// SIMATIC S7-200 SMART project (STEP 7-Micro/WIN SMART), CPU ST20

SYMBOL_TABLE 系统符号
Always_On        SM0.0    // 始终接通
First_Scan_On    SM0.1    // 仅在第一个扫描周期时接通
END_SYMBOL_TABLE

ORGANIZATION_BLOCK MAIN:OB1
TITLE=// ============================================================
// // 文件: OB1_MAIN.stl
// // 功能: PLC主循环程序
// // 项目: 药液配置与加注控制系统
// // Story: AQEX-6 状态机骨架 + AQEX-9 急停调度顺序确认
// // PLC: S7-200 SMART CPU ST20
// // 说明: 本文件为语句表(STL)格式，可参考导入STEP 7-Micro/WIN SMART
// // 调度顺序: FC0(初始化)→FC2(急停,最高优先级)→FC4(Modbus)→FC3(报警)→FC22(RTC同步)
// //           →FC1(状态调度)
// //           FC2在FC1之前,保证急停触发时同周期转S_ERROR
// // ============================================================
// 
// // 符号注释（实际导入时在符号表定义）
// // VW2     : 状态机当前状态 (0=S0,1=S1...8=S7,99=ERROR)
// // VW4     : 注射泵状态码
// // VW6     : 当前最高优先级报警码
// // VW8     : 实验轮次计数
// // V0.0    : CMD_Start (HMI→PLC启动命令)
// // V0.2    : CMD_Stop  (HMI→PLC停止命令)
// // V1.0    : STA_StartAck (PLC→HMI启动确认)
// // I1.1    : DI_EStop (急停反馈，常闭，ON=正常)
// // I0.3    : DI_Btn_SystemReset (系统复位按钮)
// 
// 
BEGIN
Network 1
//  首次扫描初始化
//  SM0.1仅在首次扫描周期ON，调用FC0系统初始化
LD     First_Scan_On:SM0.1
=      L60.0                 // 局部存储器中转
LD     L60.0
CALL   SysInit:SBR0




Network 2
//  急停与安全处理（每周期调用，优先级最高）
//  SM0.0常ON，每周期调用FC2
LD     Always_On:SM0.0
CALL   EStopHandling:SBR2




Network 3
//  HMI停止命令(V0.2) - 自动运行中任意状态可停止
//  ★ 2026-09-11 修复:
//    (1) 去掉 AW< VW2, 99 条件,允许 S_ERROR 态(VW2=99)也能停止
//        原逻辑只允许 VW2=1~8 停止, S_ERROR 锁死时点停止被忽略
//        新逻辑: VW2>0(非S0)就能停止, 急停/继电器故障锁存位由 FC19 管理
//    (2) 补清阀门诊断子状态 VB260~VB275 和诊断计时器 T50~T55
//        原三个清理路径(停止/冷启动/复位)全部遗漏,导致
//        FC11/FC15/FC17 的 AW=VW2xx,0 前置条件不成立,
//        开阀指令被跳过,表现为"点启动 M10.2=1 但系统不运行"
LD     V0.2
EU
AW>    VW2, 0                // VW2>0(排除S0), VW2=1~8 或 99 都允许停止
LPS
R      CPU_输出0:Q0.0, 7       // 泵停/阀关/NC电磁阀失电
R      T37, 1                // 停S1计时器
R      M10.2, 1              // 清S1首次进入标志
R      M10.7, 1              // 清预规划标志
R      M11.6, 1              // 清注射泵写请求
// ★ 新增: 清阀门诊断子状态+结果(VB260~VB275, 8字=16字节)
 // ★ 新增: 清阀门诊断子状态+结果(VB260~VB275, 8字=16字节)
//   覆盖: 阀A子状态VB260~261, 阀B子状态VB262~263,
 //   覆盖: 阀A子状态VB260~261, 阀B子状态VB262~263,
//         阀A/B结果VB266~269, 阀C诊断VB270~273, 其他辅助变量
 //         阀A/B结果VB266~269, 阀C诊断VB270~273, 其他辅助变量
FILL   0, VW260, 8
// ★ 新增: 清阀A/B诊断计时器 T50~T55
 // ★ 新增: 清阀A/B诊断计时器 T50~T55
R      T50, 6
MOVW   0, VW2                // 回S0
R      V0.2, 1               // 清停止命令
LPP




Network 4
//  Modbus通讯轮询（每周期调用）
LD     Always_On:SM0.0
CALL   ModbusPolling:SBR4




Network 5
//  报警处理（每周期调用）
LD     Always_On:SM0.0
CALL   AlarmHandling:SBR3




Network 6
//  RTC时间同步处理（每周期调用）
//  处理HMI校时命令V0.6和5分钟超时保护
LD     Always_On:SM0.0
CALL   RTC_Sync:SBR24




Network 7
//  状态机调度（急停时FC2会强制VW2=99）
//  每周期根据VW2调用对应状态FC
LD     Always_On:SM0.0
CALL   StateDispatcher:SBR1




Network 8
//  实验轮次计数（S5每完成一轮S1→S6累加）
//  简化骨架：在S6完成转S5时累加，实际在FC17中处理
//  此处预留，具体在FC17实现
Network 9
//  手动控制处理（仅在S0态调用,在状态调度之后）
//  处理HMI画面3手动控制命令位V306.0~V307.1
//    (旧地址V2.4~V3.5因与VW2物理重叠已于2026-09-03迁移,详见FC20符号表)
//  由FC20使用M13.0~M13.4锁存输出,NC电磁阀自动跟随(详见FC20)
LD     Always_On:SM0.0
LDW=   VW2, 0
CALL   ManualControl:SBR15




Network 10
//  手动注射泵控制（仅在S0态调用,在手动阀门控制之后）
//  处理V307.2/V307.3命令位
//    (旧地址V3.6/V3.7因与VW2物理重叠已于2026-09-03迁移,详见FC21符号表)
//  由FC21使用VD384/VW388/VW390执行单次/循环抽排(详见FC21)
LD     Always_On:SM0.0
LDW=   VW2, 0
CALL   ManualSyringePump:SBR23




Network 11
//  非S0态清除手动控制锁存与手动注射泵状态,防止返回S0时误动作
LD     Always_On:SM0.0
LDW=   VW2, 0
NOT
R      M13.0, 5              // 清阀门/泵手动锁存
R      M13.5, 3              // 清手动注射泵标志(M13.5~M13.7)
MOVW   0, VW390              // 手动注射泵子状态复位为空闲




Network 12
//  系统总状态计算 → VB305
//  优先级: 急停(2) > 故障(1) > 良好(0)
//  急停触发: I1.1=OFF(急停反馈,常闭触点断开) OR V300.4=1(急停锁存) OR V300.5=1(继电器故障)
//  故障触发: VW6<>0(有活动未确认报警) AND 非急停级
//  良好: 既非急停也无报警
//  用途: McgsPro画面顶部"良好/故障/急停"状态指示灯绑定
//  分支1: 急停级 → VB305=2
LD     CPU_输入9:I1.1          // 急停反馈(ON=正常)
NOT                          // OFF=急停触发
O      V300.4                // 或急停锁存
O      V300.5                // 或继电器故障
MOVB   2, VB305              // 急停条件满足时写2


// 分支2: 非急停 且 有活动报警 → VB305=1
 // 分支2: 非急停 且 有活动报警 → VB305=1
LDN    CPU_输入9:I1.1          // 急停已释放
AN     V300.4                // 且急停锁存=0
AN     V300.5                // 且继电器故障=0
LDW<>  VW6, 0                // 且有活动报警码
ALD                          // 合并"非急停"与"有报警"
MOVB   1, VB305              // 故障条件满足时写1


// 分支3: 非急停 且 无报警 → VB305=0
 // 分支3: 非急停 且 无报警 → VB305=0
LDN    CPU_输入9:I1.1          // 急停已释放
AN     V300.4                // 且急停锁存=0
AN     V300.5                // 且继电器故障=0
LDW=   VW6, 0                // 且无活动报警码
ALD                          // 合并"非急停"与"无报警"
MOVB   0, VB305              // 良好条件满足时写0




// ============================================================
 // ============================================================
// 文件结束
                     // 文件结束
// 说明:
                      // 说明:
//   1. FC0/FC1/FC2/FC3/FC4 见各自独立文件
 //   1. FC0/FC1/FC2/FC3/FC4 见各自独立文件
//   2. FC10~FC19 各状态FC见 State_Sxx.stl 文件
 //   2. FC10~FC19 各状态FC见 State_Sxx.stl 文件
//   3. FC20 手动控制(新增,AQEX-34修复)
 //   3. FC20 手动控制(新增,AQEX-34修复)
//   4. FC22 RTC时间同步处理(新增,AQEX-51)
 //   4. FC22 RTC时间同步处理(新增,AQEX-51)
//   5. 导入时需先建符号表，再逐个新建FC并粘贴代码
 //   5. 导入时需先建符号表，再逐个新建FC并粘贴代码
//   6. VB305 系统状态字(=0良好/1故障/2急停,AQEX-50新增)
 //   6. VB305 系统状态字(=0良好/1故障/2急停,AQEX-50新增)
// ============================================================
 // ============================================================


END_ORGANIZATION_BLOCK

SUBROUTINE_BLOCK SysInit:SBR0
TITLE=// ============================================================
// // 文件: FC0_SysInit.stl
// // 功能: 系统初始化（首次扫描SM0.1调用）
// // Story: AQEX-6 状态机骨架 + AQEX-11 断电保持与恢复逻辑
// // 说明: 双路径初始化:
// //   冷启动(V304.0=0): 全部清零安全状态,转S0
// //   断电恢复(V304.0=1): RTC检测+VD_S5_Elapsed重算+状态机恢复策略
// //   阀门动作态(S1~S6)断电 → 转S_ERROR(安全)
// //   S5(实验运行)断电 → 重算Elapsed,保持S5继续
// // 修复记录:
// //   2026-09-04: 合并所有 JMP/LBL 到单一 NETWORK，修复跨 NETWORK 跳转导致
// //               STOP/RUN 时 S0 被误判为动作态转 S_ERROR 的问题。
// //               S_ERROR 状态无实际故障时转 S0，避免历史遗留错误锁定。
// //   2026-09-04: 增加 DT10 合法性检查，避免历史垃圾时间戳误触发 RTC 丢失。
// //   2026-09-04: RTC 异常时改为置位 V303.7 请求 HMI 校时，不再直接转 S_ERROR；
// //               5 分钟未同步由 FC22 超时后进 S_ERROR 并置 V303.5。
// //   2026-09-05: 注射泵复位目标地址 40003 改用 16#9C43，避免 MOVD 十进制大数
// //               被解析为 INT 导致 MBUS_MSG Error=6。
// // ============================================================
// 
// // 符号说明:
// // V304.0: M_InitDone        初始化完成标志(断电保持,首次成功后置1)
// // VW198 : VW_Init_Step      初始化步骤号(调试用,0=完成)
// // VD186 : VD_RTC_Now_Sec    当前RTC转换总秒数(BCD转秒)
// // VD190 : VD_DT10_Sec       DT10转换总秒数(BCD转秒)
// // VD194 : VD_RTC_DT_Diff    RTC与DT10秒数差
// // V1.7  : M_TankB_State     下缸状态(1=满,断电恢复时判断是否重算Elapsed)
// // V303.5: M_Alarm_RTC_Lost  RTC时钟丢失报警(超时未同步后置位)
// // V303.7: M_Need_RTC_Sync  请求HMI同步PLC时间
// // V0.6  : CMD_RTC_Sync     HMI校时命令(上升沿触发)
// // DT10  : VB10~VB17         下缸变满时间戳(BCD)
// // RTC   : VB900~VB907       READ_RTC读取结果(BCD)
// 
// 
BEGIN
Network 1
//  步骤=1
LD     First_Scan_On:SM0.1
MOVW   1, VW198


// ★ 2026-09-07修复: 每次首次扫描(STOP→RUN/上电)统一清零Modbus库存储区和状态
 // ★ 2026-09-07修复: 每次首次扫描(STOP→RUN/上电)统一清零Modbus库存储区和状态
//   原因: 断电恢复路径(V304.0=1)不清库存储区,残留库状态机导致MBUS_MSG报Error=6
 //   原因: 断电恢复路径(V304.0=1)不清库存储区,残留库状态机导致MBUS_MSG报Error=6
//   不区分冷启动/断电恢复,统一清零(库状态机在STOP→RUN后必须复位)
 //   不区分冷启动/断电恢复,统一清零(库状态机在STOP→RUN后必须复位)
LD     First_Scan_On:SM0.1
FILL   0, VW600, 143         // VB600~VB885清零(Modbus库存储区)
LD     First_Scan_On:SM0.1
MOVB   0, VB378              // 清MBUS_CTRL Error
LD     First_Scan_On:SM0.1
MOVB   0, VB379              // 清MBUS_MSG Error(注射泵状态)
LD     First_Scan_On:SM0.1
MOVB   0, VB380              // 清MBUS_MSG Error(流量计)
LD     First_Scan_On:SM0.1
MOVB   0, VB381              // 清MBUS_MSG Error(注射泵位置)
LD     First_Scan_On:SM0.1
R      M10.0, 6              // 清M10.0~M10.5(Done位/降级标志)
LD     First_Scan_On:SM0.1
R      M11.0, 1              // 清MBUS_CTRL Done位
LD     First_Scan_On:SM0.1
MOVW   0, VW390              // 清手动注射泵子状态(防止断电恢复时残留旧值导致误触发回零)
LD     First_Scan_On:SM0.1
R      M11.6, 1              // 清注射泵写请求(防止断电恢复时残留)
LD     First_Scan_On:SM0.1
R      T104, 1               // 清回零冷却定时器
LD     First_Scan_On:SM0.1
MOVW   0, VW516              // 清FC21监控计数器
LD     First_Scan_On:SM0.1
MOVW   0, VW518
LD     First_Scan_On:SM0.1
MOVW   0, VW520
LD     First_Scan_On:SM0.1
MOVW   0, VW522
LD     First_Scan_On:SM0.1
MOVW   0, VW524
LD     First_Scan_On:SM0.1
MOVW   0, VW526
LD     First_Scan_On:SM0.1
MOVW   0, VW528
LD     First_Scan_On:SM0.1
MOVW   0, VW530
LD     First_Scan_On:SM0.1
MOVW   0, VW532
LD     First_Scan_On:SM0.1
MOVW   0, VW534
LD     First_Scan_On:SM0.1
MOVW   0, VW536
LD     First_Scan_On:SM0.1
MOVW   0, VW538
LD     First_Scan_On:SM0.1
MOVW   0, VW540
LD     First_Scan_On:SM0.1
MOVW   0, VW542
LD     First_Scan_On:SM0.1
MOVW   0, VW544
LD     First_Scan_On:SM0.1
MOVW   0, VW546
LD     First_Scan_On:SM0.1
MOVW   0, VW548


// 判断冷启动/断电恢复
               // 判断冷启动/断电恢复
LD     V304.0
JMP    1                     // V304.0=1 → 断电恢复路径


// ========== 冷启动路径 ==========
 // ========== 冷启动路径 ==========
LD     First_Scan_On:SM0.1
AN     V304.0                // 冷启动(V304.0=0)


// 注射泵单步分辨率(25ml注射器标准6000步模式)
 // 注射泵单步分辨率(25ml注射器标准6000步模式)
MOVR   4.1667, VD350         // VD_StepResolution


// ---- HMI设定参数默认值（冷启动安全初始化） ----
 // ---- HMI设定参数默认值（冷启动安全初始化） ----
// 出厂/长期断电后,HMI未配置时也有合理默认值,防止全0导致TON立即超时
 // 出厂/长期断电后,HMI未配置时也有合理默认值,防止全0导致TON立即超时


// 6.1 浓度与容量参数  ? v2.0 删除: 浓度参数整体移除, VD10~VD17 让给 DT10 RTC 独占
 // 6.1 浓度与容量参数  ? v2.0 删除: 浓度参数整体移除, VD10~VD17 让给 DT10 RTC 独占
//    原 VD10=目标浓度、VD14=母液浓度, 加药量改为用户直接输入 VD370
 //    原 VD10=目标浓度、VD14=母液浓度, 加药量改为用户直接输入 VD370


// 6.2 时间周期参数
               // 6.2 时间周期参数
MOVR   30.0, VD354           // VD_CycleSetpoint 换水周期(min)
MOVR   480.0, VD24           // VD_ExperimentTarget 实验总时长(min)
MOVR   120.0, VD28           // VD_PreMixTime S2预循环标称时长(s)
MOVR   30.0, VD32            // VD_PreMixTime_MinSafe S2压缩下限(s)
MOVR   60.0, VD36            // VD_RestTime S3.5静止等候标称时长(s)
MOVR   15.0, VD40            // VD_RestTime_Min S3.5压缩下限(s)
MOVR   5.0, VD44             // VD_CycleExtend_Max 换水周期顺延最大幅度(min)
MOVR   300.0, VD144          // VD_T_Default 首轮配液总时长默认值(s)
MOVR   180.0, VD108          // VD_S6_Default 首轮S6排水时长默认值(s)


// 6.2.1 工艺目标参数
             // 6.2.1 工艺目标参数
MOVR   10.0, VD316           // 目标进水量(L,默认10L)
MOVR   5000.0, VD370         // ? v2.0 新增: VD_Vol_Target 默认加药量(μL,默认5mL)
                          // 浓度参数删除后 VD370 改为 HMI 直接输入,需安全默认值防止全0导致 FC13 加药量=0
 // 浓度参数删除后 VD370 改为 HMI 直接输入,需安全默认值防止全0导致 FC13 加药量=0


// 6.3 超时保护参数(关键!防止TON PT=0立即超时)
 // 6.3 超时保护参数(关键!防止TON PT=0立即超时)
MOVR   60.0, VD358           // VD_Timeout_ValveA 阀A开/关到位超时(s)
MOVR   60.0, VD362           // VD_Timeout_ValveB 阀B开/关到位超时(s)
MOVR   60.0, VD54            // VD_Timeout_ValveC 阀C开/关到位超时(s)
MOVR   10.0, VD58            // VD_Timeout_Pump1 (预留未用)
MOVR   10.0, VD62            // VD_Timeout_Pump2 (预留未用)
MOVR   5.0, VD66             // VD_Delay_ValveA_Verify 阀A关后延时验证(s)


// 7.4 其他超时阈值
               // 7.4 其他超时阈值
MOVR   1800.0, VD448         // VD_S4WaitTimeout S4等待超时阈值(s,默认30min)
MOVR   10000.0, VD452        // VD_ManualDose_Target 手动总加药量(μL,默认10mL) ← 出厂硬编码
MOVW   0, VW388              // VW_ManualDose_Mode 手动模式(0=单次,1=循环) ← 出厂硬编码


// ============================================================
 // ============================================================
// v2.0 新增: 用户默认参数覆盖 (出厂默认先跑一遍,再用用户默认覆盖)
 // v2.0 新增: 用户默认参数覆盖 (出厂默认先跑一遍,再用用户默认覆盖)
// 安全兜底: 出厂硬编码永远保留,用户默认存断电保持区
 // 安全兜底: 出厂硬编码永远保留,用户默认存断电保持区
// V区分配:
                    // V区分配:
//   VB456 = 用户默认有效标志 (0=出厂默认 / 1=用户自定义)
 //   VB456 = 用户默认有效标志 (0=出厂默认 / 1=用户自定义)
//   VD460~VD528 = 18 个 REAL 用户存储 (72字节)
 //   VD460~VD528 = 18 个 REAL 用户存储 (72字节)
//   VB532 = VW388 低字节用户默认 (ManualDose_Mode)
 //   VB532 = VW388 低字节用户默认 (ManualDose_Mode)
//   VB536 = V200.0 用户默认 (AlarmAckMode bit0)
 //   VB536 = V200.0 用户默认 (AlarmAckMode bit0)
// 标签: LBL 8 = 用户默认覆盖入口, LBL 9 = 覆盖后汇合, LBL 10 = S V200.0
 // 标签: LBL 8 = 用户默认覆盖入口, LBL 9 = 覆盖后汇合, LBL 10 = S V200.0
// ============================================================
 // ============================================================
LDB=   VB456, 1              // VB456 == 1 (用户默认有效)?
JMP    8                     // 是 → 跳 LBL 8 执行用户默认覆盖
LD     Always_On:SM0.0       // 强制 C0=1 (SM0.0 常 ON)
JMP    9                     // 无条件跳 LBL 9 (跳过覆盖,用出厂默认)


LBL    8                     // ====== 用户默认覆盖区 ======
// --- 18 个 REAL ---
        // --- 18 个 REAL ---
MOVR   VD460, VD24           // VD_ExperimentTarget 实验总时长(min)
MOVR   VD464, VD28           // VD_PreMixTime S2预循环标称时长(s)
MOVR   VD468, VD32           // VD_PreMixTime_MinSafe S2压缩下限(s)
MOVR   VD472, VD36           // VD_RestTime S3.5静止等候标称时长(s)
MOVR   VD476, VD40           // VD_RestTime_Min S3.5压缩下限(s)
MOVR   VD480, VD44           // VD_CycleExtend_Max 换水周期顺延最大幅度(min)
MOVR   VD484, VD54           // VD_Timeout_ValveC 阀C超时(s)
MOVR   VD488, VD66           // VD_Delay_ValveA_Verify 阀A关后延时(s)
MOVR   VD492, VD108          // VD_S6_Default 首轮S6排水时长(s)
MOVR   VD496, VD144          // VD_T_Default 首轮配液总时长(s)
MOVR   VD500, VD316          // VD_TargetInletVolume 目标进水量(L)
MOVR   VD504, VD350          // VD_StepResolution 脉冲当量
MOVR   VD508, VD354          // VD_CycleSetpoint 换水周期(min)
MOVR   VD512, VD358          // VD_Timeout_ValveA 阀A超时(s)
MOVR   VD516, VD362          // VD_Timeout_ValveB 阀B超时(s)
MOVR   VD520, VD370          // VD_Vol_Target 目标加药量(μL)
MOVR   VD524, VD448          // VD_S4WaitTimeout S4等待超时(s)
MOVR   VD528, VD452          // VD_ManualDose_Target 手动总加药量(μL)


// --- WORD: VW388 ManualDose_Mode (MOVW 要求源=16位,拆成两个字节) ---
 // --- WORD: VW388 ManualDose_Mode (MOVW 要求源=16位,拆成两个字节) ---
MOVB   VB532, VB388          // 复制低字节
MOVB   0, VB389              // 高字节清零


// --- BIT: V200.0 AlarmAckMode (VB536 bit0=1 则置 V200.0) ---
 // --- BIT: V200.0 AlarmAckMode (VB536 bit0=1 则置 V200.0) ---
LDB=   VB536, 1
JMP    10                    // VB536 == 1 → 跳去 S V200.0
R      V200.0, 1             // VB536 != 1 → 清 V200.0
LD     Always_On:SM0.0       // 强制 C0=1 (SM0.0 常 ON)
JMP    9                     // 无条件跳汇合点
LBL    10
S      V200.0, 1             // VB536 == 1 → 置 V200.0


LBL    9                     // ====== 覆盖后汇合点,继续初始化 ======


// 状态机初始化为S0
                // 状态机初始化为S0
MOVW   0, VW2                // VW2=0(S0)
// ★ 2026-09-11 新增: 冷启动也清阀门诊断子状态和计时器
 // ★ 2026-09-11 新增: 冷启动也清阀门诊断子状态和计时器
// 保险: 即使冷启动,VB260~VB275可能残留断电前状态,
 // 保险: 即使冷启动,VB260~VB275可能残留断电前状态,
// 导致下次启动FC11/FC15/FC17的AW=VW2xx,0前置条件不成立
 // 导致下次启动FC11/FC15/FC17的AW=VW2xx,0前置条件不成立
FILL   0, VW260, 8           // 清 VB260~VB275 (阀A/B/C 诊断)
R      T50, 6                // 清 T50~T55 (阀A/B 诊断计时器)
R      V1.6, 1               // 上缸=空
R      V1.7, 1               // 下缸=空


// 复位所有DO输出(安全状态)
           // 复位所有DO输出(安全状态)
MOVB   0, QB0                // Q0.0~Q0.7=0(泵停/阀关/NC电磁阀失电)
MOVB   0, QB8                // Q8.0~Q8.7=0(DR32输出全清零,含报警灯)


// 清除急停锁存
                   // 清除急停锁存
R      V300.4, 1             // M_EStop_Latch=0


// 清除报警字和报警码
                // 清除报警字和报警码
FILL   0, VW300, 4           // VB300~VB303清零(报警字)
MOVW   0, VW6                // VW6=0(无报警)


// 清除FC3内部继电器(消音/新报警检测)
     // 清除FC3内部继电器(消音/新报警检测)
R      M11.1, 1              // M_Sound_Latched=0(消音标志)
R      M11.2, 1              // M_PrevAlarm=0(上周期有报警标志)


// ★ 2026-09-06新增(FC99调试经验): 清空Modbus库存储区VB600~VB885
 // ★ 2026-09-06新增(FC99调试经验): 清空Modbus库存储区VB600~VB885
//   V区断电不丢,残留的库状态机会导致MBUS_MSG报Error=6(忙)
 //   V区断电不丢,残留的库状态机会导致MBUS_MSG报Error=6(忙)
//   库分配: Modbus RTU Master (v2.0) → VB600~VB885(286字节=143字)
 //   库分配: Modbus RTU Master (v2.0) → VB600~VB885(286字节=143字)
FILL   0, VW600, 143         // VB600~VB885清零(Modbus库存储区)


// ★ 2026-09-11修复: 冷启动必须清 VB0, 防止 V0.x 命令位断电保持后卡1
 // ★ 2026-09-11修复: 冷启动必须清 VB0, 防止 V0.x 命令位断电保持后卡1
//   现场现象: V0.3(CMD_AckAlarm)卡在1 → FC3 Network 4 EU无上升沿 → R V0.3,1 永远不执行
 //   现场现象: V0.3(CMD_AckAlarm)卡在1 → FC3 Network 4 EU无上升沿 → R V0.3,1 永远不执行
//   V0.x 是 HMI→PLC 的脉冲命令, FC3/OB1/FC10 会在收到后自清除, 冷启动清0无副作用
 //   V0.x 是 HMI→PLC 的脉冲命令, FC3/OB1/FC10 会在收到后自清除, 冷启动清0无副作用
MOVB   0, VB0                // V0.0~V0.7 全部清0
// 清除命令握手位
                  // 清除命令握手位
R      V1.0, 6               // V1.0~V1.5=0


// 实验轮次清零
                   // 实验轮次清零
MOVW   0, VW8                // VW8=0


// 本次实验累计流量清零
               // 本次实验累计流量清零
MOVR   0.0, VD364            // VD_ExpTotal_Flow=0(L)


// 本次实验累计加药量清零
              // 本次实验累计加药量清零
MOVR   0.0, VD440            // VD_Dosed_Volume_Total=0(μL)


// S4等待时长清零(内部变量,每次S4完成也会清)
 // S4等待时长清零(内部变量,每次S4完成也会清)
MOVR   0.0, VD444            // ? v2.0 新增: VD_S4Wait_Time 冷启动清零


// S3剩余待加药量清零
               // S3剩余待加药量清零
MOVR   0.0, VD372            // VD_Remaining_Vol=0(μL)


// 清下缸满计时器+预规划标志
            // 清下缸满计时器+预规划标志
MOVR   0.0, VD178            // VD_S5_Elapsed=0
R      M10.7, 1              // 清预规划触发标志


// 初始化Modbus轮询计数器与状态
        // 初始化Modbus轮询计数器与状态
// 注意:VW250/VW252与HMI参数VD250重叠,已迁移到VW290/VW292/VW294/VW296/VW504
 // 注意:VW250/VW252与HMI参数VD250重叠,已迁移到VW290/VW292/VW294/VW296/VW504
MOVW   0, VW290              // 轮询计数器=0(任务0)
MOVW   0, VW292              // 任务0(注射泵状态)连续失败计数=0
MOVW   0, VW294              // 任务1(流量计)连续失败计数=0
MOVW   0, VW296              // 任务2(注射泵位置)连续失败计数=0
MOVW   0, VW504              // 任务2(注射泵位置)成功计数=0
R      M10.0, 6              // 清M10.0~M10.5(Done位/降级标志)
LD     First_Scan_On:SM0.1
R      T103, 1               // 清MBUS_MSG超时定时器
LD     First_Scan_On:SM0.1
S      M15.0, 1              // 首次扫描启动任务0(注射泵状态)
LD     First_Scan_On:SM0.1
R      M15.1, 1              // 清任务1/2使能标志
LD     First_Scan_On:SM0.1
R      M15.2, 1
R      V60.0, 6              // 清V60.0~V60.5(FC4/FC21/FC3中间继电器)
R      M11.0, 1              // 清MBUS_CTRL Done位
R      M11.6, 1              // 清注射泵写请求
R      M11.7, 1              // 清注射泵写忙
R      M12.0, 1              // 清注射泵写完成
R      V304.1, 1             // 清注射泵在线标志(冷启动后由FC4实时刷新)
R      V304.2, 1             // 清流量计在线标志(冷启动后由FC4实时刷新)
R      M12.1, 1              // 清S3抽液开始标志
R      M12.2, 1              // 清S3排液开始标志
R      M13.0, 5              // 清手动控制锁存(M13.0~M13.4),防止STOP→RUN后误输出
R      M13.5, 3              // 清手动注射泵标志(M13.5~M13.7)
MOVW   0, VW390              // 手动注射泵子状态=0(空闲)
MOVR   0.0, VD392            // 手动累计加药量=0(内部)
MOVR   0.0, VD396            // 手动剩余加药量=0(内部)


// 手动注射泵参数已移至出厂硬编码阶段(L142~L143),此处不再重复
 // 手动注射泵参数已移至出厂硬编码阶段(L142~L143),此处不再重复
// 否则会覆盖用户默认值 (Bug fix 2026-09-12)
 // 否则会覆盖用户默认值 (Bug fix 2026-09-12)
MOVB   0, VB378              // 清MBUS_CTRL Error
MOVB   0, VB379              // 清MBUS_MSG Error(注射泵状态)
MOVB   0, VB380              // 清MBUS_MSG Error(流量计)
MOVB   0, VB381              // 清MBUS_MSG Error(注射泵位置)
MOVB   0, VB382              // 清MBUS_MSG Error(瞬时流量)
MOVB   0, VB383              // 清MBUS_MSG Error(写命令)
MOVR   0.0, VD374            // 流量计降级值清零
MOVW   0, VW226              // 清S3子状态
MOVD   0, VD232              // 清写目标地址
MOVW   0, VW230              // 清写数据


// ★ 2026-09-06修正: 冷启动不再自动下发注射泵复位
 // ★ 2026-09-06修正: 冷启动不再自动下发注射泵复位
// 原因: FC99现场调试确认, 泵上电后默认进入96(就绪态), 可直接接受命令
 // 原因: FC99现场调试确认, 泵上电后默认进入96(就绪态), 可直接接受命令
//       无需复位; 且自动复位会在泵未就绪时发送命令, 可能导致103错误
 //       无需复位; 且自动复位会在泵未就绪时发送命令, 可能导致103错误
//       如需复位, 由HMI手动触发或S3加药流程按需触发
 //       如需复位, 由HMI手动触发或S3加药流程按需触发
LD     First_Scan_On:SM0.1
AN     V304.0
MOVD   0, VD232              // 清写目标地址(不自动复位)
MOVW   0, VW230              // 清写数据
R      M11.6, 1              // 确保写请求位清零


MOVW   2, VW198              // 步骤=2(冷启动完成)
JMP    2                     // → 完成


// ========== 断电恢复路径 ==========
 // ========== 断电恢复路径 ==========
// ★ Story1.7 决策9: 报警位断电恢复处理 — 断电保持区报警位保持,FC0不主动清除
 // ★ Story1.7 决策9: 报警位断电恢复处理 — 断电保持区报警位保持,FC0不主动清除
//   (由FC3/FC19按确认流程处理)。断电前已触发的报警仍需人工确认;仅冷启动才清报警字。
 //   (由FC3/FC19按确认流程处理)。断电前已触发的报警仍需人工确认;仅冷启动才清报警字。
LBL    1
LD     First_Scan_On:SM0.1
TODR   VB900                 // 读RTC到VB900~VB907(BCD)
// 注: 断电恢复路径不清 VW300~303/VW6/V300.x 等报警位, 让FC3 NETWORK1每周期重算
 // 注: 断电恢复路径不清 VW300~303/VW6/V300.x 等报警位, 让FC3 NETWORK1每周期重算
//   操作员重新上电后能看到断电前未处理的报警,按正常流程确认清除
 //   操作员重新上电后能看到断电前未处理的报警,按正常流程确认清除


// RTC自身合法性检查(RTC字段越界→请求校时)
 // RTC自身合法性检查(RTC字段越界→请求校时)
LDB>   VB901, 12             // 月>12
JMP    4
LDB<   VB901, 1              // 月<1
JMP    4
LDB>   VB902, 31             // 日>31
JMP    4
LDB<   VB902, 1              // 日<1
JMP    4
LDB>   VB903, 23             // 时>23
JMP    4
LDB>   VB904, 59             // 分>59
JMP    4
LDB>   VB905, 59             // 秒>59
JMP    4


// RTC丢失检测: 比较RTC与DT10(VB10~VB17)
 // RTC丢失检测: 比较RTC与DT10(VB10~VB17)
// DT10未写入(VB10=0)→跳过检测
     // DT10未写入(VB10=0)→跳过检测
LDB=   VB10, 0
JMP    3


// DT10数据合法性检查（防止历史垃圾数据误触发RTC丢失）
 // DT10数据合法性检查（防止历史垃圾数据误触发RTC丢失）
LDB<   VB11, 1               // 月<1
JMP    4
LDB>   VB11, 12              // 月>12
JMP    4
LDB<   VB12, 1               // 日<1
JMP    4
LDB>   VB12, 31              // 日>31
JMP    4
LDB>   VB13, 23              // 时>23
JMP    4
LDB>   VB14, 59              // 分>59
JMP    4
LDB>   VB15, 59              // 秒>59
JMP    4


// 逐字段BCD比较(年→月→日→时→分→秒)
    // 逐字段BCD比较(年→月→日→时→分→秒)
LDB<   VB900, VB10           // RTC年 < DT10年 → RTC丢失
JMP    4
LDB>   VB900, VB10           // RTC年 > DT10年 → 正常
JMP    3
LDB<   VB901, VB11           // 比月
JMP    4
LDB>   VB901, VB11
JMP    3
LDB<   VB902, VB12           // 比日
JMP    4
LDB>   VB902, VB12
JMP    3
LDB<   VB903, VB13           // 比时
JMP    4
LDB>   VB903, VB13
JMP    3
LDB<   VB904, VB14           // 比分
JMP    4
LDB>   VB904, VB14
JMP    3
LDB<   VB905, VB15           // 比秒
JMP    4
LD     Always_On:SM0.0       // 全部>= → RTC正常
JMP    3


// RTC异常/丢失 → 请求HMI校时
       // RTC异常/丢失 → 请求HMI校时
LBL    4
LD     First_Scan_On:SM0.1
S      V303.7, 1             // M_Need_RTC_Sync
MOVR   0.0, VD178            // VD_S5_Elapsed=0(无法重算)
MOVW   3, VW198              // 步骤=3(RTC需校时)
JMP    5                     // → 状态恢复


// RTC正常，继续
                 // RTC正常，继续
LBL    3
MOVW   3, VW198              // 步骤=3(RTC正常)


// BCD转秒 - RTC(VD_RTC_Now_Sec)
 // BCD转秒 - RTC(VD_RTC_Now_Sec)
LD     First_Scan_On:SM0.1
MOVR   0.0, VD186            // 清VD_RTC_Now_Sec
BTI    VB903, AC0            // BCD→INT(时)
ITD    AC0, AC0              // INT→DINT
DTR    AC0, AC0              // DINT→REAL
*R     3600.0, AC0           // ×3600
+R     AC0, VD186            // 累加到VD_RTC_Now_Sec
BTI    VB904, AC0            // 分
ITD    AC0, AC0
DTR    AC0, AC0
*R     60.0, AC0
+R     AC0, VD186
BTI    VB905, AC0            // 秒
ITD    AC0, AC0
DTR    AC0, AC0
+R     AC0, VD186


// BCD转秒 - DT10(VD_DT10_Sec)
 // BCD转秒 - DT10(VD_DT10_Sec)
LD     First_Scan_On:SM0.1
MOVR   0.0, VD190            // 清VD_DT10_Sec
BTI    VB13, AC0             // DT10时
ITD    AC0, AC0
DTR    AC0, AC0
*R     3600.0, AC0
+R     AC0, VD190
BTI    VB14, AC0             // 分
ITD    AC0, AC0
DTR    AC0, AC0
*R     60.0, AC0
+R     AC0, VD190
BTI    VB15, AC0             // 秒
ITD    AC0, AC0
DTR    AC0, AC0
+R     AC0, VD190
MOVW   4, VW198              // 步骤=4(BCD转秒完成)


// VD_S5_Elapsed重算(仅保持S5且下缸=满时)
 // VD_S5_Elapsed重算(仅保持S5且下缸=满时)
LD     V1.7                  // 下缸=满
AW=    VW2, 6                // 且状态机=S5(字比较,与栈顶AND)
MOVR   VD186, VD178          // 满足:VD_S5_Elapsed = RTC秒
-R     VD190, VD178          // - DT10秒 = 断电期间经过秒数
MOVW   5, VW198              // 步骤=5(Elapsed重算完成)
JMP    5                     // → 状态恢复


// 下缸=空 或 非S5 时VD_S5_Elapsed=0
 // 下缸=空 或 非S5 时VD_S5_Elapsed=0
LD     Always_On:SM0.0
MOVR   0.0, VD178            // Elapsed=0
MOVW   5, VW198


// 状态机恢复策略
                  // 状态机恢复策略
LBL    5
LDW=   VW2, 0
JMP    6                     // S0保持
LDW=   VW2, 6
JMP    6                     // S5保持(断电续跑)
LDW=   VW2, 8
JMP    6                     // S7保持(锁定态)


// S_ERROR: 无实际故障则转S0，否则保持
  // S_ERROR: 无实际故障则转S0，否则保持
LDW=   VW2, 99
JMP    7


// S1~S6: 阀门/泵动作中断 → 转S_ERROR
 // S1~S6: 阀门/泵动作中断 → 转S_ERROR
LD     Always_On:SM0.0
MOVB   0, QB0                // 阀门关/泵停/NC电磁阀失电(安全)
MOVW   99, VW2               // 转S_ERROR
S      V300.4, 1             // 置急停锁存(类比急停,需人工复位)
MOVW   7, VW198              // 步骤=7(状态机转S_ERROR)
JMP    2


// S_ERROR特殊处理
              // S_ERROR特殊处理
LBL    7
LD     V300.4                // 急停锁存
O      V300.5                // 或继电器故障
O      CPU_输入9:I1.1          // 或急停触发
LDW<>  VW6, 0                // 或有活动报警
OLD
JMP    6                     // 任一满足 → 保持S_ERROR


// 无实际故障 → 转S0
              // 无实际故障 → 转S0
LD     First_Scan_On:SM0.1
MOVB   0, QB0                // 输出安全状态
R      CPU_输出7:Q0.7, 1       // 清报警声音
MOVW   0, VW2                // 转S0
MOVW   6, VW198              // 步骤=6(状态恢复完成)
JMP    2


// 保持原状态
                    // 保持原状态
LBL    6
MOVW   6, VW198              // 步骤=6(状态恢复完成)


// ========== 初始化完成 ==========
 // ========== 初始化完成 ==========
LBL    2
LD     First_Scan_On:SM0.1
S      V304.0, 1             // M_InitDone=1(初始化完成,断电保持)
MOVW   0, VW198              // 步骤=0(完成)




// 注: 冷启动(V304.0=0)时全部清零+HMI设定参数初始化为安全默认值
 // 注: 冷启动(V304.0=0)时全部清零+HMI设定参数初始化为安全默认值
// 注: 断电恢复(V304.0=1)时保留断电保持数据(含用户HMI设定值)
 // 注: 断电恢复(V304.0=1)时保留断电保持数据(含用户HMI设定值)
// 注: 阀门动作态(S1~S6)断电转S_ERROR,因阀门状态未知(可能半开),强制安全
 // 注: 阀门动作态(S1~S6)断电转S_ERROR,因阀门状态未知(可能半开),强制安全
// 注: S5(实验运行)断电可恢复,无阀门动作,VD_S5_Elapsed由RTC重算连续不跳变
 // 注: S5(实验运行)断电可恢复,无阀门动作,VD_S5_Elapsed由RTC重算连续不跳变
// 注: RTC丢失(RTC<DT10)触发V303.5,转S_ERROR,需HMI校时后人工复位
 // 注: RTC丢失(RTC<DT10)触发V303.5,转S_ERROR,需HMI校时后人工复位
// 注: BCD转秒用当天秒数(时×3600+分×60+秒),跨天场景需补天数×86400
 // 注: BCD转秒用当天秒数(时×3600+分×60+秒),跨天场景需补天数×86400
// 注: S_ERROR无实际故障(V300.4/5=0,I1.1=0,VW6=0)时转S0,避免历史遗留锁定
 // 注: S_ERROR无实际故障(V300.4/5=0,I1.1=0,VW6=0)时转S0,避免历史遗留锁定




// ============================================================
 // ============================================================
// 文件结束
                     // 文件结束
// ============================================================
 // ============================================================


END_SUBROUTINE_BLOCK

SUBROUTINE_BLOCK StateDispatcher:SBR1
TITLE=// ============================================================
// // 文件: FC1_StateDispatcher.stl
// // 功能: 状态机调度器（每周期根据VW2调用对应状态FC）
// // Story: AQEX-6 状态机骨架
// // 说明: S7-200 SMART STL无CASE语句，用比较+跳转实现
// // 修复记录:
// //   P1-NETWORK标题去掉冒号(错误66)
// //   P2-JMP/LBL跨NETWORK问题修复: 全部合并到NETWORK 1
// // ============================================================
// 
BEGIN
Network 1
//  状态调度 (JMP/LBL必须在同一NETWORK内)
//  读取VW2并与各状态值比较，相等则调用对应FC
//  VW2 = 0 → S0初始化
LDW<=  VW2, 0
JMP    1


// VW2 = 1 → S1上缸进水
         // VW2 = 1 → S1上缸进水
LDW=   VW2, 1
JMP    2


// VW2 = 2 → S2预循环
          // VW2 = 2 → S2预循环
LDW=   VW2, 2
JMP    3


// VW2 = 3 → S3加药
           // VW2 = 3 → S3加药
LDW=   VW2, 3
JMP    4


// VW2 = 4 → S3.5静止等候
       // VW2 = 4 → S3.5静止等候
LDW=   VW2, 4
JMP    5


// VW2 = 5 → S4上→下转移
        // VW2 = 5 → S4上→下转移
LDW=   VW2, 5
JMP    6


// VW2 = 6 → S5实验运行中
        // VW2 = 6 → S5实验运行中
LDW=   VW2, 6
JMP    7


// VW2 = 7 → S6下缸排水
         // VW2 = 7 → S6下缸排水
LDW=   VW2, 7
JMP    8


// VW2 = 8 → S7实验结束
         // VW2 = 8 → S7实验结束
LDW=   VW2, 8
JMP    9


// VW2 = 99 → S_ERROR故障锁定
   // VW2 = 99 → S_ERROR故障锁定
LDW=   VW2, 99
JMP    10


// 其他非法值 → 强制回S0
            // 其他非法值 → 强制回S0
LDW>=  VW2, 100
JMP    11


// 若未匹配任何状态(0<VW2<99但非上述值)，也回S0
 // 若未匹配任何状态(0<VW2<99但非上述值)，也回S0
JMP    11


// S0入口
                     // S0入口
LBL    1
CALL   State_S0_Init:SBR5
JMP    12


// S1入口
                     // S1入口
LBL    2
S      M10.2, 1              // S1首次进入脉冲
CALL   State_S1_Inlet:SBR6
JMP    12


// S2入口
                     // S2入口
LBL    3
CALL   State_S2_PreMix:SBR7
JMP    12


// S3入口
                     // S3入口
LBL    4
CALL   State_S3_Dosing:SBR8
JMP    12


// S3.5入口
                   // S3.5入口
LBL    5
CALL   State_S35_Rest:SBR9
JMP    12


// S4入口
                     // S4入口
LBL    6
CALL   State_S4_Transfer:SBR10
JMP    12


// S5入口
                     // S5入口
LBL    7
CALL   State_S5_Run:SBR11
JMP    12


// S6入口
                     // S6入口
LBL    8
CALL   State_S6_Drain:SBR12
JMP    12


// S7入口
                     // S7入口
LBL    9
CALL   State_S7_End:SBR13
JMP    12


// S_ERROR入口
                // S_ERROR入口
LBL    10
CALL   State_Error:SBR14
JMP    12


// 非法状态处理（强制回S0）
            // 非法状态处理（强制回S0）
LBL    11
MOVW   0, VW2                // VW2=0


// 调度结束
                     // 调度结束
LBL    12
// 状态调度完成，返回OB1
             // 状态调度完成，返回OB1




// ============================================================
 // ============================================================
// 文件结束
                     // 文件结束
// 说明:
                      // 说明:
//   1. JMP/LBL必须在同一NETWORK内(修复跨网络跳转问题)
 //   1. JMP/LBL必须在同一NETWORK内(修复跨网络跳转问题)
//   2. 每个状态FC内部负责状态转移(修改VW2)
 //   2. 每个状态FC内部负责状态转移(修改VW2)
//   3. 修复VW2=1无法保持的问题(原跨NETWORK跳转导致程序流混乱)
 //   3. 修复VW2=1无法保持的问题(原跨NETWORK跳转导致程序流混乱)
// ============================================================
 // ============================================================


END_SUBROUTINE_BLOCK

SUBROUTINE_BLOCK EStopHandling:SBR2
TITLE=// ============================================================
// // 文件: FC2_EStopHandling.stl
// // 功能: 急停与安全处理（每周期调用，优先级最高）
// // Story: AQEX-6 状态机骨架 + AQEX-9 急停双通道+安全继电器反馈(详细实现)
// // 说明: 急停检测(I1.1 上升沿:NO 闭合)→锁存V300.4→转S_ERROR  v1.3 NO 进 I1.1
// //       安全继电器反馈延时校验(2秒)→V300.5继电器故障最高级报警
// //       输出强制安全(QB0=0,Q0.7声音开)
// //       急停解除与系统复位由FC19(State_Error)处理
// // ============================================================
// 
// // 符号说明:
// // I1.1  : DI_EStop           急停反馈(常开 NO,OFF=正常,ON=急停触发)  v1.3 改为接 NO 触点
// // I1.2  : DI_SafetyRelay_FB  安全继电器辅助反馈(ON=动力回路接通,OFF=动力回路断开)
// // V300.4: M_EStop_Latch      急停触发锁存(漫溢级,强制人工确认)
// // V300.5: M_Alarm_SafetyRelay 安全继电器故障(最高级,强制人工确认)
// // VW2   : 状态机状态(FC2写99转S_ERROR)
// // VW6   : 报警码(99=继电器故障,10=急停)
// // T35   : 安全继电器反馈延时(PT=20,2秒)
// // M10.7 : 预规划触发标志(急停时清,防止S5残留)
BEGIN
Network 1
//  急停触发检测(I1.1 上升沿) + 锁存 + 转S_ERROR  v1.3: NO 进 PLC,上升沿触发
//  I1.1接常开 NO:OFF=正常,ON=急停触发 (v1.3 NC 改去 MSR-P,NO 进 PLC I1.1)
//  NO 触点按下时 I1.1 变 ON,EU 上升沿检测"按下瞬间"
LD     CPU_输入9:I1.1
EU
S      V300.4, 1             // M_EStop_Latch锁存
MOVW   99, VW2               // VW2=99(转S_ERROR)
// 清预规划标志(防止S5残留干扰)
         // 清预规划标志(防止S5残留干扰)
R      M10.7, 1




Network 2
//  安全继电器反馈延时校验
//  急停锁存后,2秒内I1.2应反馈"动力回路已断开"(I1.2=OFF)
//  I1.2定义:ON=动力回路接通(辅助触点反馈),OFF=动力回路已断开
//  若2秒后I1.2仍ON → 主触点可能粘连,继电器故障
LD     V300.4                // 急停已锁存
A      CPU_输入10:I1.2         // 且动力回路仍接通(未确认断开)
TON    T35, 20               // 2秒延时(20×100ms)


LD     T35                   // 延时到达
EU
S      V300.5, 1             // M_Alarm_SafetyRelay(最高级报警)




Network 3
//  急停锁存时输出强制安全
//  急停锁存时,每周期强制QB0=0(泵停/阀关/NC电磁阀失电=安全)
//  Q0.7报警声音开(急停立即报警)
//  Q8.0灯光不在此处理,由FC3报警处理统一管理(避免双写冲突)
LD     V300.4                // M_EStop_Latch
MOVB   0, QB0                // 潜水泵停/阀A/B/C关/NC电磁阀失电(关闭=安全)
S      CPU_输出7:Q0.7, 1       // 报警声音开




Network 4
//  报警码写入(优先级:继电器故障99 > 急停10)
LD     V300.5                // 继电器故障(最高级)
MOVW   99, VW6               // VW6=99
JMP    1


LD     V300.4                // 急停(无继电器故障)
AN     V300.5
MOVW   10, VW6               // VW6=10


LBL    1




// 注: 急停解除与系统复位逻辑在FC19(State_Error)中处理
 // 注: 急停解除与系统复位逻辑在FC19(State_Error)中处理
// 注: Q8.0报警灯光由FC3 AlarmHandling按VW6优先级统一管理(Story 1.6)
 // 注: Q8.0报警灯光由FC3 AlarmHandling按VW6优先级统一管理(Story 1.6)
// 注: I1.2接线逻辑:ON=动力回路接通,OFF=动力回路断开(与代码注释一致)
 // 注: I1.2接线逻辑:ON=动力回路接通,OFF=动力回路断开(与代码注释一致)
// 注: 安全继电器反馈延时2秒兼顾机械动作时间与故障捕获灵敏度
 // 注: 安全继电器反馈延时2秒兼顾机械动作时间与故障捕获灵敏度
// 注: 急停硬件回路(安全继电器切断动力电)不经过PLC,本FC仅处理软件层面
 // 注: 急停硬件回路(安全继电器切断动力电)不经过PLC,本FC仅处理软件层面




// ============================================================
 // ============================================================
// 文件结束
                     // 文件结束
// ============================================================
 // ============================================================


END_SUBROUTINE_BLOCK

SUBROUTINE_BLOCK AlarmHandling:SBR3
TITLE=// ============================================================
// // 文件: FC3_AlarmHandling.stl
// // 功能: 报警处理（每周期调用）
// // Story: AQEX-6 状态机骨架 + AQEX-10 报警分级与消音/消光逻辑(详细实现)
// // 说明: 优先级链计算VW6 + 消音(I0.4/V0.4) + 消光(V0.3确认)
// //       自动恢复模式(V200.0=0时一般故障级条件消失自动复位)
// //       高优先级(漫溢/节奏滞后/继电器故障)强制人工确认,不受模式影响
// // ============================================================
// 
// // 符号说明:
// // VW6   : 当前最高优先级未确认报警码(0=无,99=继电器故障,10~14漫溢,20~21节奏,30~65一般)
// // V200.0: M_AlarmAckMode 报警确认模式(0=自动恢复,1=人工确认)
// // Q0.7  : 报警声音(FC2/FC19置位,FC3管理消音)
// // Q8.0  : 报警灯光(FC3统一管理,避免双写冲突)
// // I0.4  : 就地消音按钮(常开点动)
// // V0.3  : CMD_AckAlarm HMI报警确认命令
// // V0.4  : CMD_Mute HMI消音命令
// // V1.3  : STA_AlarmAckDone 报警确认握手
// // V1.4  : STA_MuteDone 消音握手
// // M11.1 : M_Sound_Latched 声音已消音标志(新报警时清,实现重鸣)
// // M11.2 : M_PrevAlarm 上一周期有报警标志(新报警检测用)
// 
// 
BEGIN
Network 1
//  优先级链计算VW6(最高优先级未确认报警码)
//  优先级: 99 > 10~14 > 20 > 21 > 30~36 > 40~47 > 60~65
//  用LD压栈+条件JMP实现,JMP nAlarmCodeDone跳到末尾
//  最高级: 安全继电器故障
LD     V300.5
JMP    1


// 漫溢级(10~14)
               // 漫溢级(10~14)
LD     V300.0
JMP    2
LD     V300.1
JMP    3
LD     V300.2
JMP    4
LD     V300.3
JMP    5
LD     V300.4
JMP    6


// 节奏滞后级(20~21)
             // 节奏滞后级(20~21)
LD     V300.6
JMP    7
LD     V300.7
JMP    8


// 阀A类(30~36)
               // 阀A类(30~36)
LD     V301.0
JMP    9
LD     V301.1
JMP    10
LD     V301.2
JMP    11
LD     V301.3
JMP    12
LD     V301.4
JMP    13
LD     V301.5
JMP    14
LD     V301.6
JMP    15


// 阀B/C/泵类(40~47)
           // 阀B/C/泵类(40~47)
LD     V302.0
JMP    16
LD     V302.1
JMP    17
LD     V302.2
JMP    18
LD     V302.3
JMP    19
LD     V302.4
JMP    20
LD     V302.5
JMP    21
LD     V302.6
JMP    22
LD     V302.7
JMP    23


// 其他(60~65)
                // 其他(60~65)
LD     V303.0
JMP    24
LD     V303.1
JMP    25
LD     V303.2
JMP    26
// ★ 2026-09-11修复: V303.3 为预留未使用位,不再映射报警码(与故障代码字典/报警字映射表对齐)
 // ★ 2026-09-11修复: V303.3 为预留未使用位,不再映射报警码(与故障代码字典/报警字映射表对齐)
LD     V303.4
JMP    28
LD     V303.5
JMP    29


// 无报警
                      // 无报警
LD     Always_On:SM0.0
MOVW   0, VW6
JMP    31


// 报警码赋值
                    // 报警码赋值
LBL    1
MOVW   99, VW6
JMP    31
LBL    2
MOVW   10, VW6
JMP    31
LBL    3
MOVW   11, VW6
JMP    31
LBL    4
MOVW   12, VW6
JMP    31
LBL    5
MOVW   13, VW6
JMP    31
LBL    6
MOVW   14, VW6
JMP    31
LBL    7
MOVW   20, VW6
JMP    31
LBL    8
MOVW   21, VW6
JMP    31
LBL    9
MOVW   30, VW6
JMP    31
LBL    10
MOVW   31, VW6
JMP    31
LBL    11
MOVW   32, VW6
JMP    31
LBL    12
MOVW   33, VW6
JMP    31
LBL    13
MOVW   34, VW6
JMP    31
LBL    14
MOVW   35, VW6
JMP    31
LBL    15
MOVW   36, VW6
JMP    31
LBL    16
MOVW   40, VW6
JMP    31
LBL    17
MOVW   41, VW6
JMP    31
LBL    18
MOVW   42, VW6
JMP    31
LBL    19
MOVW   43, VW6
JMP    31
LBL    20
MOVW   44, VW6
JMP    31
LBL    21
MOVW   45, VW6
JMP    31
LBL    22
MOVW   46, VW6
JMP    31
LBL    23
MOVW   47, VW6
JMP    31
LBL    24
MOVW   60, VW6
JMP    31
LBL    25
MOVW   61, VW6
JMP    31
LBL    26
// ★ 2026-09-11修复: V303.2 正确报警码是 49(S4转移等待超时), 之前错写成 62
 // ★ 2026-09-11修复: V303.2 正确报警码是 49(S4转移等待超时), 之前错写成 62
MOVW   49, VW6
JMP    31
// ★ 2026-09-11修复: 删掉 LBL 27(V303.3=预留未使用位, 无报警码)
 // ★ 2026-09-11修复: 删掉 LBL 27(V303.3=预留未使用位, 无报警码)
LBL    28
MOVW   64, VW6
JMP    31
LBL    29
MOVW   65, VW6


LBL    31




Network 2
//  报警输出管理(灯光常亮 + 新报警声音重鸣)
//  有活动报警(VW6≠0) → 灯光Q8.0常亮
//  新报警(VW6由0变非0) → 清M_Sound_Latched,声音重鸣
LDW<>  VW6, 0
S      EM0_输出0:Q8.0, 1       // 灯光常亮


// 新报警检测: 本周期VW6≠0 且 上一周期M11.2=0(无报警) → 新报警
 // 新报警检测: 本周期VW6≠0 且 上一周期M11.2=0(无报警) → 新报警
LDW<>  VW6, 0
AN     M11.2                 // 上一周期无报警 → 新报警
R      M11.1, 1              // 清消音标志(新报警重鸣)


// 声音管理: 有报警且未消音 → 声音开
      // 声音管理: 有报警且未消音 → 声音开
LDW<>  VW6, 0
AN     M11.1                 // 未消音
S      CPU_输出7:Q0.7, 1       // 声音开


// 自动恢复模式: VW6=0且自动模式 → 自动消光
 // 自动恢复模式: VW6=0且自动模式 → 自动消光
LDW=   VW6, 0
AN     V200.0                // M_AlarmAckMode=0(自动模式)
R      EM0_输出0:Q8.0, 1       // 无报警自动消光
R      CPU_输出7:Q0.7, 1       // 无报警关声音
R      M11.1, 1              // 清消音标志


// 更新上一周期报警标志
               // 更新上一周期报警标志
LDW<>  VW6, 0
=      M11.2                 // 记录本周期有报警(供下周期新报警检测)




Network 3
//  消音处理(I0.4就地按钮 OR V0.4 HMI命令)
//  消音源: I0.4上升沿 OR V0.4上升沿
LD     CPU_输入4:I0.4
EU
LD     V0.4
EU
OLD                          // 两者任一上升沿
R      CPU_输出7:Q0.7, 1       // 关声音
S      M11.1, 1              // 置消音标志(新报警时清)
S      V1.4, 1               // STA_MuteDone握手
R      V0.4, 1               // 清HMI消音命令
// 注: 消音只关声音,灯光Q8.0和报警位保持;新报警(VW6变化)时M11.1清,声音重鸣
 // 注: 消音只关声音,灯光Q8.0和报警位保持;新报警(VW6变化)时M11.1清,声音重鸣




Network 4
//  报警确认处理(V0.3 HMI确认 → 条件消失才消光+清锁存)
//  V0.3上升沿 = HMI报警确认命令(高优先级HMI侧二次确认,PLC只收V0.3)
//  确认规则: V0.3上升沿后,逐个检查报警位条件,条件消失的复位报警位,再由NETWORK1重算VW6
//  ★ 关键修复(2026-09-04): NETWORK 4 缺 V0.3 上升沿门控(JMP),导致每周期无条件
//    执行所有条件复位,包括 LD V303.5; R V303.5, 1——使 S_ERROR 立即被清
//    修复: V0.3 无上升沿时跳过整个网络,避免误清报警位
//  ★★★ 2026-09-11 发现 JMP 条件写反了！ ★★★
//    原代码 LD V0.3; EU; JMP 40：EU=1(有上升沿)时跳转 → 反而跳过了 R V0.3,1
//    正确：用 V60.5 缓存 EU 结果,LDN 取反后触发 JMP,再用 LD 恢复栈顶执行线圈
//    注意：STL 的 S/R/= 线圈指令依赖栈顶=1 才执行,不能用 NOT+JMP（会清掉栈顶）
//    注意：S7-200 SMART 不支持 JMPN 指令,必须用 JMP + LDN 中转
LD     V0.3
EU
=      V60.5                 // 缓存 EU 结果: 有上升沿=1, 无上升沿=0
LDN    V60.5                 // 无上升沿时栈顶=1
JMP    40                    // ★ 无上升沿则跳转到 LBL 40,跳过确认处理
LD     V60.5                 // 有上升沿时栈顶=1,恢复执行条件


S      V1.3, 1               // STA_AlarmAckDone握手
R      V0.3, 1               // 清确认命令


// 漫溢级: 条件消失才复位(液位计高位=OFF)
  // 漫溢级: 条件消失才复位(液位计高位=OFF)
LD     V300.0                // 上缸漫溢
AN     CPU_输入5:I0.5          // 液位计A-高位已OFF
R      V300.0, 1             // 复位
LD     V300.1                // 下缸漫溢
AN     CPU_输入7:I0.7          // 液位计B-高位已OFF
R      V300.1, 1
// NC阀动作: 由人工确认复位(无DI直接条件,保持锁存需HMI强制,此处不自动复位)
 // NC阀动作: 由人工确认复位(无DI直接条件,保持锁存需HMI强制,此处不自动复位)
// 急停V300.4/继电器故障V300.5: 由FC19系统复位按钮/HMI高权限确认处理,FC3不碰
 // 急停V300.4/继电器故障V300.5: 由FC19系统复位按钮/HMI高权限确认处理,FC3不碰


// 节奏滞后级: 条件消失(新一轮开始)由FC40重置,FC3不直接处理
 // 节奏滞后级: 条件消失(新一轮开始)由FC40重置,FC3不直接处理
// 但V0.3确认时,若V300.6/7已由FC40清除,NETWORK1会重算VW6
 // 但V0.3确认时,若V300.6/7已由FC40清除,NETWORK1会重算VW6


// 一般故障级: 条件消失则复位
           // 一般故障级: 条件消失则复位
// 阀A类
                      // 阀A类
LD     V301.0                // 阀A关后仍有流
AN     CPU_输入0:I0.0          // 流量开关A已OFF
R      V301.0, 1
LD     V301.1                // 阀A内漏
AN     CPU_输入0:I0.0          // 流量开关A已OFF
R      V301.1, 1
LD     V301.2                // 阀A关到位超时
A      EM0_输入1:I8.1          // 阀A关到位反馈已ON
R      V301.2, 1
LD     V301.3                // 阀A关到位但仍有流
AN     CPU_输入0:I0.0          // 流量开关A已OFF
R      V301.3, 1
LD     V301.4                // 阀A开到位超时
A      EM0_输入0:I8.0          // 阀A开到位反馈已ON
R      V301.4, 1
LD     V301.5                // 阀A开到位但无流
A      CPU_输入0:I0.0          // 流量开关A已ON
R      V301.5, 1
LD     V301.6                // S5触发S1时上缸≠空
AN     V1.6                  // 上缸已=空
R      V301.6, 1


// 阀B/C类
                    // 阀B/C类
LD     V302.0                // 阀B诊断异常
LD     CPU_输入1:I0.1          // 流量开关B=ON(已恢复)
O      CPU_输入6:I0.6          // 或液位计A-低位=ON
ALD
R      V302.0, 1
LD     V302.1                // 阀B开到位超时
A      EM0_输入2:I8.2
R      V302.1, 1
LD     V302.2                // 阀B开到位但无流
A      CPU_输入1:I0.1
R      V302.2, 1
LD     V302.3                // 阀B关到位超时
A      EM0_输入3:I8.3
R      V302.3, 1
LD     V302.4                // 阀B关到位但仍有流
AN     CPU_输入1:I0.1
R      V302.4, 1
LD     V302.5                // 阀C诊断异常
LD     CPU_输入2:I0.2
O      CPU_输入8:I1.0
ALD
R      V302.5, 1
LD     V302.6                // 阀C开到位超时
A      EM0_输入4:I8.4
R      V302.6, 1
LD     V302.7                // 阀C开到位但无流
A      CPU_输入2:I0.2
R      V302.7, 1


// 其他类
                      // 其他类
LD     V303.0                // 阀C关到位超时
A      EM0_输入5:I8.5
R      V303.0, 1
LD     V303.1                // 阀C关到位但仍有流
AN     CPU_输入2:I0.2
R      V303.1, 1
LD     V303.4                // 注射泵通讯异常
AW=    VW4, 0                // 状态码=0(空闲正常)
R      V303.4, 1
LD     V303.5                // RTC时钟丢失
R      V303.5, 1             // 由HMI校时后手动确认清除


LBL    40                    // ★ NETWORK 4 跳转目标(无V0.3上升沿时跳过确认处理)


// 注: 报警位复位后,下一周期NETWORK1重算VW6;若VW6=0,NETWORK2自动消光
 // 注: 报警位复位后,下一周期NETWORK1重算VW6;若VW6=0,NETWORK2自动消光
// 注: 漫溢级(V300.2/3 NC阀)、急停(V300.4)、继电器故障(V300.5)不由FC3复位
 // 注: 漫溢级(V300.2/3 NC阀)、急停(V300.4)、继电器故障(V300.5)不由FC3复位
//      由FC19系统复位按钮/HMI高权限确认处理
 //      由FC19系统复位按钮/HMI高权限确认处理




Network 5
//  自动恢复模式(M_AlarmAckMode=0时一般故障级条件消失自动复位)
//  自动模式: V200.0=0时,一般故障级报警位条件消失自动R复位
//  漫溢/节奏滞后/继电器故障不受此模式影响,保持锁存
//  ★ 2026-09-11 修复 AQEX-XX: 状态机已进S_ERROR(VW2=99)时禁止自动清报警位
//    原因: 一般故障触发MOVW 99,VW2后，若自动恢复立即清报警位，
//    会导致 VW2=99 + VW6=0 的状态机/报警系统不一致
//    场景: 阀A开到位超时(V301.4)后阀A终于开到位(I8.0=ON),
//          FC3 NETWORK 5 自动清V301.4→VW6=0,但VW2已锁99无人解锁,
//          OB1 NETWORK12 按VW6=0算VB305=0(良好),掩盖故障
//    防御: S_ERROR态暂停自动恢复,让FC19 NETWORK5自动解锁或人工复位处理
LDW=   VW2, 99
JMP    50                    // S_ERROR态 → 跳过自动恢复,报警位保持


LD     V200.0                // M_AlarmAckMode
NOT                          // =0(自动模式)时执行后续


// 阀A类自动复位(条件消失)
            // 阀A类自动复位(条件消失)
LD     V301.0
AN     CPU_输入0:I0.0
R      V301.0, 1
LD     V301.1
AN     CPU_输入0:I0.0
R      V301.1, 1
LD     V301.2
A      EM0_输入1:I8.1
R      V301.2, 1
LD     V301.3
AN     CPU_输入0:I0.0
R      V301.3, 1
LD     V301.4
A      EM0_输入0:I8.0
R      V301.4, 1
LD     V301.5
A      CPU_输入0:I0.0
R      V301.5, 1
LD     V301.6
AN     V1.6
R      V301.6, 1


// 阀B/C类自动复位
                // 阀B/C类自动复位
LD     V302.0
LD     CPU_输入1:I0.1
O      CPU_输入6:I0.6
ALD
R      V302.0, 1
LD     V302.1
A      EM0_输入2:I8.2
R      V302.1, 1
LD     V302.2
A      CPU_输入1:I0.1
R      V302.2, 1
LD     V302.3
A      EM0_输入3:I8.3
R      V302.3, 1
LD     V302.4
AN     CPU_输入1:I0.1
R      V302.4, 1
LD     V302.5
LD     CPU_输入2:I0.2
O      CPU_输入8:I1.0
ALD
R      V302.5, 1
LD     V302.6
A      EM0_输入4:I8.4
R      V302.6, 1
LD     V302.7
A      CPU_输入2:I0.2
R      V302.7, 1


// 其他类自动复位
                  // 其他类自动复位
LD     V303.0
A      EM0_输入5:I8.5
R      V303.0, 1
LD     V303.1
AN     CPU_输入2:I0.2
R      V303.1, 1
LD     V303.4
AW=    VW4, 0
R      V303.4, 1
// V303.5(RTC丢失)不自动清除,需HMI校时后确认
 // V303.5(RTC丢失)不自动清除,需HMI校时后确认


LBL    50                    // ★ S_ERROR态跳过自动恢复的跳转目标(2026-09-11新增)


// 注: 漫溢(V300.0~3)、急停(V300.4)、继电器故障(V300.5)、节奏滞后(V300.6/7)不在此处理
 // 注: 漫溢(V300.0~3)、急停(V300.4)、继电器故障(V300.5)、节奏滞后(V300.6/7)不在此处理
// 注: 自动复位后下一周期NETWORK1重算VW6,NETWORK2自动消光
 // 注: 自动复位后下一周期NETWORK1重算VW6,NETWORK2自动消光




Network 6
//  报警日志(新报警触发时写入,简化版)
//  新报警: 本周期VW6≠0 且 上一周期M11.2=0
//  简化: 仅记录报警码和时间戳到固定位置(完整环形缓冲区由HMI侧轮询读取)
LDW<>  VW6, 0
AN     M11.2                 // 上一周期无报警 → 新报警
EU
TODR   VB500                 // 时间戳写入VB500~507
MOVB   VB7, VB509            // 报警码(VW6低字节VB7)
MOVB   1, VB510              // 动作=1(触发)
MOVB   1, VB508              // 单元编号=1(本PLC)
// 注: 完整环形缓冲区(6条×16字节)用指针AR1实现,本简化版固定VB500起
 // 注: 完整环形缓冲区(6条×16字节)用指针AR1实现,本简化版固定VB500起
// 注: 详细历史记录由HMI侧存储,PLC仅保留最新一条供HMI轮询
 // 注: 详细历史记录由HMI侧存储,PLC仅保留最新一条供HMI轮询




// ============================================================
 // ============================================================
// 文件结束
                     // 文件结束
// 说明:
                      // 说明:
//   1. FC3每周期调用,负责报警码计算+输出管理+确认处理+自动恢复+日志
 //   1. FC3每周期调用,负责报警码计算+输出管理+确认处理+自动恢复+日志
//   2. 报警位置位由各FC(FC2/FC30~32/FC40等)负责,FC3只复位
 //   2. 报警位置位由各FC(FC2/FC30~32/FC40等)负责,FC3只复位
//   3. Q8.0灯光由FC3统一管理,FC2/FC19不操作Q8.0(避免双写)
 //   3. Q8.0灯光由FC3统一管理,FC2/FC19不操作Q8.0(避免双写)
//   4. Q0.7声音由FC2/FC19置位(急停/故障态),FC3管理消音+新报警重鸣
 //   4. Q0.7声音由FC2/FC19置位(急停/故障态),FC3管理消音+新报警重鸣
//   5. 编址修正: M_AlarmAckMode=V200.0(避VD124冲突),SafetyRelayAck=V0.7(避V0.5冲突)
 //   5. 编址修正: M_AlarmAckMode=V200.0(避VD124冲突),SafetyRelayAck=V0.7(避V0.5冲突)
//   6. 高优先级(漫溢/节奏滞后/继电器故障)强制人工确认,不受M_AlarmAckMode影响
 //   6. 高优先级(漫溢/节奏滞后/继电器故障)强制人工确认,不受M_AlarmAckMode影响
//   7. NETWORK4/5的报警位复位条件需与各FC置位条件严格对应(现场调试时核实)
 //   7. NETWORK4/5的报警位复位条件需与各FC置位条件严格对应(现场调试时核实)
// ============================================================
 // ============================================================


END_SUBROUTINE_BLOCK

SUBROUTINE_BLOCK ModbusPolling:SBR4
TITLE=
BEGIN
Network 1
//   MBUS_CTRL: 9600/8/N/1, 超时1000ms
LD     Always_On:SM0.0
=      L60.0
LD     Always_On:SM0.0
=      L63.7
LD     L60.0
CALL   MBUS_CTRL:SBR20, L63.7, 9600, 16#0, 16#0, 1000, M11.0, VB378
Network 2
//   T103: MBUS_MSG超时定时器(100ms时基, PT=100=10s)
//   任一任务活跃(M15.0~M15.4)时计时, 超时后强制切换任务
LD     M15.0
O      M15.1
O      M15.2
O      M15.3
O      M15.4
TON    T103, 100
Network 3
//   任务0: 注射泵状态读(41001)
//   EN=VW290==0 AND M15.0, First=M15.0上升沿(EU)
LDW=   VW290, 0
=      L60.0
LD     M15.0
EU
=      L63.7
LD     L60.0
CALL   MBUS_MSG:SBR21, L63.7, 16#1, 16#0, 16#A029, 16#1, &VB410, M10.0, VB379
Network 4
//   任务1: 流量计读(40009)
//   EN=VW290==1 AND M15.1, First=M15.1上升沿(EU)
LDW=   VW290, 1
=      L60.0
LD     M15.1
EU
=      L63.7
LD     L60.0
CALL   MBUS_MSG:SBR21, L63.7, 16#2, 16#0, 16#9C49, 16#2, &VB410, M14.0, VB380
Network 5
//   任务2: 注射泵位置读(41007)
//   EN=VW290==2 AND M15.2, First=M15.2上升沿(EU)
LDW=   VW290, 2
=      L60.0
LD     M15.2
EU
=      L63.7
LD     L60.0
CALL   MBUS_MSG:SBR21, L63.7, 16#1, 16#0, 16#A02F, 16#1, &VB410, M10.1, VB381
Network 6
//   任务3: 流量计瞬时流量读(40007) → VD94
//   EN=VW290==3 AND M15.3, First=M15.3上升沿(EU)
LDW=   VW290, 3
=      L60.0
LD     M15.3
EU
=      L63.7
LD     L60.0
CALL   MBUS_MSG:SBR21, L63.7, 16#2, 16#0, 16#9C47, 16#2, &VB410, M14.1, VB382
Network 7
//   任务0成功处理: VW410->VW4, 成功计数, 清失败计数
LD     M10.0
A      M15.0
AB=    VB379, 0
MOVW   VW410, VW224
AENO
INCW   VW500
AENO
MOVW   0, VW292
AENO
R      V303.4, 1
Network 8
LDW=   VW224, 96
MOVW   0, VW4
Network 9
LDW=   VW224, 64
MOVW   1, VW4
Network 10
LDW=   VW224, 100
MOVW   2, VW4
Network 11
LDW<>  VW224, 100
AW<>   VW224, 96
AW<>   VW224, 64
MOVW   4, VW4
Network 12
//   任务0失败计数
LD     M10.0
A      M15.0
AB<>   VB379, 0
INCW   VW292
Network 13
//   任务0完成切换(成功或T103超时)
//   R M15.0, S M15.1, 更新VW290=1, 清Done位, 清超时定时器
LD     M10.0
O      T103
R      M15.0, 1
S      M15.1, 1
MOVW   1, VW290
R      M10.0, 1
R      T103, 1
Network 14
//   任务1成功处理: VD410->VD86, 成功计数, 清失败计数
//   流量计32位浮点数据已按正确顺序存储,直接搬运即可
LD     M14.0
A      M15.1
AB=    VB380, 0
MOVD   VD410, VD86
AENO
INCW   VW502
AENO
MOVW   0, VW294
AENO
R      V303.6, 1
Network 15
//   任务1失败计数
LD     M14.0
A      M15.1
AB<>   VB380, 0
INCW   VW294
Network 16
//   任务1完成切换(成功或T103超时)
//   R M15.1, S M15.2, 更新VW290=2, 清Done位, 清超时定时器
LD     M14.0
O      T103
R      M15.1, 1
S      M15.2, 1
MOVW   2, VW290
R      M14.0, 1
R      T103, 1
Network 17
//   任务2成功处理: VW410->VW222, 成功计数, 清失败计数
LD     M10.1
A      M15.2
AB=    VB381, 0
MOVW   VW410, VW222
AENO
INCW   VW504
AENO
MOVW   0, VW296
Network 18
//   任务2失败计数
LD     M10.1
A      M15.2
AB<>   VB381, 0
INCW   VW296
Network 19
//   任务2完成切换(成功或T103超时)
//   R M15.2, S M15.3, 更新VW290=3, 清Done位, 清超时定时器
LD     M10.1
O      T103
R      M15.2, 1
S      M15.3, 1
MOVW   3, VW290
R      M10.1, 1
R      T103, 1
Network 20
//   任务3成功处理: VD410->VD94(瞬时流量), 成功计数, 清失败计数
//   流量计32位浮点数据已按正确顺序存储,直接搬运即可
LD     M14.1
A      M15.3
AB=    VB382, 0
MOVD   VD410, VD94
AENO
INCW   VW506
AENO
MOVW   0, VW298
Network 21
//   任务3失败计数
LD     M14.1
A      M15.3
AB<>   VB382, 0
INCW   VW298
Network 22
//   任务3完成切换: 有写请求 → 任务4, 否则 → 任务0
//   用V60.0做完成事件中间继电器(仅此处赋值,无冲突)
LD     M14.1
O      T103
=      V60.0
Network 23
//  // 复位任务3相关标志
LD     V60.0
R      M15.3, 1
R      M14.1, 1
R      T103, 1
Network 24
//  // 进入任务4: 有写请求(M11.6=1)
LD     V60.0
A      M11.6
S      M15.4, 1
MOVW   4, VW290
Network 25
//  // 未进入任务4则回任务0
LD     V60.0
AN     M15.4
S      M15.0, 1
MOVW   0, VW290
Network 26
LD     V60.0
EU
INCW   VW514
Network 27
//   任务4写数据准备: 有写请求时把VW230复制到统一缓冲区VW410
//   DataPtr用&VB410, 避免直接使用&VW230导致MBUS_MSG写失败(Error=104)
LD     M11.6
MOVW   VW230, VW410
Network 28
LD     M12.0
EU
INCW   VW512
Network 29
//   任务4: 注射泵写命令(仅在M11.6=1时执行)
//   EN=VW290==4 AND M15.4 AND M11.6, First=M15.4上升沿(EU)
//   写目标地址VD232由FC0/FC13/FC21设置(16#9C42=40002强停,16#9C43=40003复位,16#9C46=40006抽液,16#9C47=40007排液)
LDW=   VW290, 4
A      M15.4
A      M11.6
=      V60.3
Network 30
LD     V60.3
=      L60.0
LD     V60.3
EU
=      L63.7
LD     L60.0
CALL   MBUS_MSG:SBR21, L63.7, 16#1, 16#1, VD232, 16#1, &VB410, M12.0, VB383
Network 31
//   任务4成功处理: 清写请求, 成功计数, 清失败计数
//   ★关键: 写完成后立即清M11.6, 防止复位命令在轮询中反复写
LD     M12.0
A      M15.4
AB=    VB383, 0
R      M11.6, 1
R      M11.7, 1
INCW   VW508
MOVW   0, VW510
R      V303.4, 1
Network 32
//   任务4失败计数 + 从站异常立即报警
LD     M12.0
A      M15.4
LPS
AB<>   VB383, 0
INCW   VW510
LPP
AB>=   VB383, 101
S      V303.4, 1
Network 33
//   任务4完成切换(成功或T103超时)
//   R M15.4, S M15.0, 更新VW290=0, 清握手, 清超时定时器
//  // ★M12.0不清! 由FC13/FC21请求方清零, 否则请求方看不到写完成
LD     M12.0
O      T103
R      M11.6, 1
R      M11.7, 1
R      M15.4, 1
S      M15.0, 1
MOVW   0, VW290
R      T103, 1
Network 34
//   V303.4软件滤波: 连续读失败<5次时不报警
LDW<   VW292, 5
R      V303.4, 1
Network 35
//   V303.4写任务软件滤波: 连续写失败<5次且无从站异常时不报警
LDW<   VW510, 5
AB<    VB383, 101
R      V303.4, 1
Network 36
//   V303.6软件滤波: 连续失败<5次时不报警
LDW<   VW294, 5
R      V303.6, 1


END_SUBROUTINE_BLOCK

SUBROUTINE_BLOCK State_S0_Init:SBR5
TITLE=// ============================================================
// // 文件: FC10_State_S0_Init.stl
// // 功能: S0初始化状态 (VW2=0)
// // Story: AQEX-6 状态机骨架
// // 说明: 等待HMI启动命令，无活动报警时转S1
// // ============================================================
// 
BEGIN
Network 1
//  S0状态输出（安全待命）
//  仅复位Q0.0~Q0.6(泵/阀/NC电磁阀),Q0.7报警声音由FC3统一管理,避免本FC与FC3双写导致闪亮
LD     Always_On:SM0.0
R      CPU_输出0:Q0.0, 7       // 泵停、阀A/B/C关、NC电磁阀失电(关闭),保留Q0.7




Network 2
//  检测启动命令 - 带上缸液位前置条件
//  V0.0(CMD_Start)上升沿 AND 无活动报警(VW6=0) AND 上缸空(I0.6=ON) → 转S1
//  ★ 2026-09-11 新增硬件液位开关检查
//  原实现只查 VW6=0，遗漏了上缸必须排空才能启动的前置条件
//  用户现场: 上缸有液体(I0.6=OFF=低位开关未闭合=未排空)时点启动,
//            系统直接进S1开阀A进水,等于往未排空的缸里继续加液,与设计不符
//  为什么只查上缸(I0.6)不查下缸(I1.0):
//    S1是上缸进水阶段,只动上缸;下缸有水不影响S1的任何动作,
//    所以启动前置只卡 I0.6(上缸排空)即可,下缸状态在S4/S6阶段各自互锁
//  为什么用硬件开关而不是软件V1.6:
//    V1.6/V1.7 是软件标志,冷启动/复位时被 FC0 强制复位为1(空),
//    是假阳性;必须用硬件液位开关 I0.6(NPN常闭,液体低于探针闭合=I=1=上缸排空)
//  启动条件:
//    V0.0↑        — 用户点启动
//    AND VW6=0    — 无活动报警(FC3管理)
//    AND I0.6=ON  — 上缸排空(NPN常闭低液位,闭合=液体低于探针)
// 
//  STL实现说明: MOVR/MOVW/FILL/S/R 都是无条件执行,不受RLO影响
//  所以不能靠 LPS 门控启动代码,必须用 JMP 跳过
//  结构:
//    EU触发 → VW6=0 → 上缸空?
//      是 → R V301.1(清旧提示) → 播种+转态 → JMP跳过报警
//      否 → JMP跳过启动代码 → S V301.7(发提示) → 继续
//    最后统一 R V0.0,1 (不管成功失败,用户每次点按钮都是独立脉冲)
LD     V0.0                  // CMD_Start
EU                           // 上升沿检测,只触发一次
LPS                          // 压栈保存 EU 结果
AW=    VW6, 0                // 无活动报警 (RLO = EU AND VW6=0)
// 检查上缸未排空的条件
               // 检查上缸未排空的条件
AN     CPU_输入6:I0.6          // 上缸未排空 (NPN常闭未闭合=液体没过探针)
JMP    1                     // 上缸未排空 → 跳 LBL 1 (跳过启动代码,去发提示)
// 上缸排空 → 执行启动代码 (JMP 未触发时才走到这)
 // 上缸排空 → 执行启动代码 (JMP 未触发时才走到这)
// ★ 顺手清掉之前可能残留的 V301.7 提示位 (方案A: 满足条件自动清除)
 // ★ 顺手清掉之前可能残留的 V301.7 提示位 (方案A: 满足条件自动清除)
R      V301.7, 1             // 启动条件已满足,旧提示清除
// 【首轮播种】滚动值初始化为HMI设定的默认值
   // 【首轮播种】滚动值初始化为HMI设定的默认值
MOVR   VD144, VD112          // T滚动值 ← T默认值(HMI设定)
MOVR   VD108, VD116          // S6滚动值 ← S6默认值(HMI设定)
// 状态转移：S0→S1
               // 状态转移：S0→S1
MOVW   1, VW2                // VW2=1(S1)
// 握手确认
                     // 握手确认
S      V1.0, 1               // STA_StartAck=1
// 启动成功 → 跳过提示代码, 直接去清启动命令
  // 启动成功 → 跳过提示代码, 直接去清启动命令
JMP    2


LBL    1                     // ← 上缸未排空时跳到这
// 发启动条件不满足提示
               // 发启动条件不满足提示
// 一般故障级, 不加进VW6优先级链, 不锁S_ERROR
 // 一般故障级, 不加进VW6优先级链, 不锁S_ERROR
// 仅HMI滚动条提示"启动条件不满足: 上缸未排空"
 // 仅HMI滚动条提示"启动条件不满足: 上缸未排空"
S      V301.7, 1


LBL    2                     // ← 启动成功/提示后都汇聚到这
// 清除启动命令位
                  // 清除启动命令位
R      V0.0, 1


LPP                          // 弹栈结束




// 注: 急停触发由FC2强制VW2=99，此处不处理
 // 注: 急停触发由FC2强制VW2=99，此处不处理
// 注: S7实验结束后HMI确认重启也走此路径(经S_ERROR解除后回S0)
 // 注: S7实验结束后HMI确认重启也走此路径(经S_ERROR解除后回S0)




// ============================================================
 // ============================================================
// 文件结束
                     // 文件结束
// ============================================================
 // ============================================================


END_SUBROUTINE_BLOCK

SUBROUTINE_BLOCK State_S1_Inlet:SBR6
TITLE=// ============================================================
// // 文件: FC11_State_S1_Inlet.stl
// // 功能: S1上缸进水 (VW2=1)
// // Story: AQEX-6 状态机骨架 + AQEX-7 阀门诊断(已集成) + AQEX-8 节奏纠偏(已集成二次校正)
// // 说明: 开阀A进水，调用FC30阀A诊断(差值法+延时验证)
// //       诊断结果VW266: 0进行中/1正常完成/2故障
// //       诊断正常完成 → 调用FC40二次校正(模式1) → 更新VD_T_Rolling → 转S2
// // ============================================================
// 
// // 符号说明:
// // VW260 : Diag_State_A  阀A诊断子状态
// // VW266 : Diag_Result_A 阀A诊断结果
// // VW278 : VD_Timeout_ValveA×10 转换值(供FC30的T50用,已修正避FC32冲突)
// // VW280 : VD_Delay_ValveA_Verify×10 转换值(供FC30的T51用)
// // VD332 : VD358运算中间变量(避免修改HMI参数VD358)
// // VD250 : 目标进水量(HMI设定)
// 
// 
BEGIN
Network 1
//  S1首次进入 - 开阀A + NC球阀 + 复位计时器
LD     M10.2
AW=    VW260, 0
S      CPU_输出2:Q0.2, 1       // 开阀A
S      CPU_输出5:Q0.5, 1       // 开上缸NC球阀
R      T37, 1                // 复位S1计时器
R      V1.6, 1               // 置上缸状态=空




Network 2
//  S1首次进入 - 流量计快照
LD     M10.2
AW=    VW260, 0
MOVD   VD86, VD82




Network 3
//  S1首次进入 - 计算超时参数 VW278 = VD358 × 10
LD     M10.2
AW=    VW260, 0
MOVR   VD358, VD332
*R     10.0, VD332
ROUND  VD332, AC0
MOVW   AC0, VW278




Network 4
//  S1首次进入 - 计算延时参数 VW280 = VD66 × 10
LD     M10.2
AW=    VW260, 0
MOVR   VD66, VD320
*R     10.0, VD320
ROUND  VD320, AC0
MOVW   AC0, VW280




Network 5
//  S1首次进入 - 启动阀A诊断(最后执行,使上方各段条件成立)
LD     M10.2
AW=    VW260, 0
MOVB   1, VB260              // 子状态=1(等待开到位)
MOVB   0, VB261
MOVB   0, VB266              // 清诊断结果
MOVB   0, VB267




Network 6
//  调用阀A诊断FC30
LD     Always_On:SM0.0
CALL   ValveA_Diag:SBR16




Network 7
//  检查阀A诊断结果 + 二次校正 + 转S2
//  VW266=0 进行中，继续等待
//  VW266=1 正常完成 → 二次校正 → 转S2
//  VW266=2 故障(FC30已转S_ERROR)，本周期结束
LD     Always_On:SM0.0
AW=    VW266, 1              // 诊断正常完成?
JMP    1                     // 是 → 跳转处理
LD     Always_On:SM0.0
JMP    2                     // 否 → 结束本NETWORK


LBL    1
LD     Always_On:SM0.0
R      T37, 1                // 停S1计时
MOVW   T37, VW414            // 暂存定时器值(16位整数)
ITD    VW414, VD444          // 整数→双整数
DTR    VD444, VD70           // 双整数→实数(VD_S1_Actual)
// 【Story1.4】二次校正(7.3): 用S1实测值重核S2/S3.5目标
 // 【Story1.4】二次校正(7.3): 用S1实测值重核S2/S3.5目标
// Available' = CycleSetpoint×60 + S6_Rolling - S5_Elapsed(已含S1耗时)
 // Available' = CycleSetpoint×60 + S6_Rolling - S5_Elapsed(已含S1耗时)
LD     Always_On:SM0.0
MOVR   VD354, VD150          // VD_CycleSetpoint(min)
*R     60.0, VD150           // →秒
+R     VD116, VD150          // + VD_S6_Rolling
-R     VD178, VD150          // - VD_S5_Elapsed = Available'
// Needed' = S2_Target(预规划已定) + S3_Estimate + RestTime_Target(预规划已定)
 // Needed' = S2_Target(预规划已定) + S3_Estimate + RestTime_Target(预规划已定)
MOVR   VD120, VD154          // VD_S2_Target
+R     VD174, VD154          // + VD_S3_Estimate
+R     VD124, VD154          // + VD_RestTime_Target = Needed'
MOVW   1, VW182              // 模式=1(二次校正)
CALL   RhythmCorrection:SBR19
// 更新VD_T_Rolling(取标称值,7.5): S1实测+S2标称+S3估算+S3.5标称
 // 更新VD_T_Rolling(取标称值,7.5): S1实测+S2标称+S3估算+S3.5标称
LD     Always_On:SM0.0
MOVR   VD70, VD112           // VD_S1_Actual
+R     VD28, VD112           // + VD_PreMixTime(S2标称)
+R     VD174, VD112          // + VD_S3_Estimate
+R     VD36, VD112           // + VD_RestTime(S3.5标称) = 新VD_T_Rolling
// 二次校正非人工介入(4) → 转S2
       // 二次校正非人工介入(4) → 转S2
LD     Always_On:SM0.0
AW<>   VW184, 4
// 累加本次进水量到本次实验累计流量
         // 累加本次进水量到本次实验累计流量
MOVR   VD90, AC0             // AC0 = VD_Current_InletVolume
+R     AC0, VD364            // VD_ExpTotal_Flow += 本次进水量
MOVW   2, VW2                // 状态转移 S1→S2
R      M10.2, 1              // 清S1首次进入标志


LBL    2




// 注: 漫溢保护、差值法计量、延时验证、内漏检测、开关到位诊断
 // 注: 漫溢保护、差值法计量、延时验证、内漏检测、开关到位诊断
//      全部由FC30统一处理，FC11仅负责状态转移调度
 //      全部由FC30统一处理，FC11仅负责状态转移调度
// 注: VD250(目标进水量)由HMI设定或FC11进入时计算
 // 注: VD250(目标进水量)由HMI设定或FC11进入时计算
// 注: 二次校正(Story 1.4)在转S2前调用
 // 注: 二次校正(Story 1.4)在转S2前调用
// 注: VD358运算已改用独立中间变量VD332,不再修改HMI设定参数
 // 注: VD358运算已改用独立中间变量VD332,不再修改HMI设定参数
// 注: 断电恢复由FC0统一处理,VW2=1(S1阀A动作中断)时FC0转S_ERROR
 // 注: 断电恢复由FC0统一处理,VW2=1(S1阀A动作中断)时FC0转S_ERROR




// ============================================================
 // ============================================================
// 文件结束
                     // 文件结束
// ============================================================
 // ============================================================


END_SUBROUTINE_BLOCK

SUBROUTINE_BLOCK State_S2_PreMix:SBR7
TITLE=// ============================================================
// // 文件: FC12_State_S2_PreMix.stl
// // 功能: S2预循环搅拌 (VW2=2)
// // Story: AQEX-6 状态机骨架 + A1修复(计时转换)
// // 说明: 开潜水泵1/2搅拌，计时到达VD_S2_Target转S3
// //       v9.4更新: 取消潜水泵1/2流量开关及超时保护(I0.3/I0.4/T44/T45)
// // ============================================================
// 
// // 符号说明:
// // VW252 : VD_S2_Target×10 转换值(100ms时基,供T38用)
// // VD336 : VD120运算中间变量(避免修改VD_S2_Target)
BEGIN
Network 1
//  S2进入动作
//  启动潜水泵1和2
LD     Always_On:SM0.0
S      CPU_输出0:Q0.0, 1       // 潜水泵1开
S      CPU_输出1:Q0.1, 1       // 潜水泵2开
// 计算T38 PT值: VW252 = VD_S2_Target(VD120) × 10 (REAL秒→100ms时基)
 // 计算T38 PT值: VW252 = VD_S2_Target(VD120) × 10 (REAL秒→100ms时基)
// A1修复: 原骨架标注"待Story1.4补充转换",FC40只输出REAL秒到VD120,
 // A1修复: 原骨架标注"待Story1.4补充转换",FC40只输出REAL秒到VD120,
//         从未写入VW252导致T38计时失效。现补转换逻辑。
 //         从未写入VW252导致T38计时失效。现补转换逻辑。
MOVR   VD120, VD336          // 复制到中间变量(避免修改VD_S2_Target)
*R     10.0, VD336
ROUND  VD336, AC0
MOVW   AC0, VW252            // VW252 = VD120×10
R      T38, 1
TON    T38, VW252            // PT=VD_S2_Target×10(100ms时基)
// 置上缸状态=满
                  // 置上缸状态=满
S      V1.6, 1




Network 2
//  预循环完成转移至S3
//  注: S3期间潜水泵继续运行(搅拌+加药同时进行),此处不停止
LD     T38                   // 计时到达
MOVW   3, VW2                // VW2=3(S3)
MOVW   0, VW226              // 清S3加药子状态




// ============================================================
 // ============================================================
// 文件结束
                     // 文件结束
// 说明:
                      // 说明:
//   1. A1修复: VW252由VD120×10转换写入(原骨架遗漏,导致T38计时失效)
 //   1. A1修复: VW252由VD120×10转换写入(原骨架遗漏,导致T38计时失效)
//   2. v9.4更新: 取消潜水泵1/2流量开关及超时保护(T44/T45/VW282/VW284/VD344不再使用)
 //   2. v9.4更新: 取消潜水泵1/2流量开关及超时保护(T44/T45/VW282/VW284/VD344不再使用)
//   3. VD336为运算中间变量,不污染HMI设定参数
 //   3. VD336为运算中间变量,不污染HMI设定参数
// ============================================================
 // ============================================================


END_SUBROUTINE_BLOCK

SUBROUTINE_BLOCK State_S3_Dosing:SBR8
TITLE=// ============================================================
// // 文件: FC13_State_S3_Dosing.stl
// // 功能: S3加药 (VW2=3)
// // Story: AQEX-6 状态机骨架 + 注射泵控制(AQEX-50)
// // 说明: 计算加药步数, 通过Modbus FC06依次下发抽液/排液指令,
// //       每次动作后发强停(40002=1)恢复96就绪态, 出错转S_ERROR
// //
// // 2026-09-06修正(基于FC99现场调试):
// //   1. 地址格式: 40006→16#9C46, 40007→16#9C47, 40002→16#9C42
// //   2. 状态码: VW4=0(96就绪), VW4=1(64空闲), VW4=2(100运动中), VW4≥4(错误)
// //   3. 强停恢复: 每次抽液/排液运动完成后发强停(40002=1)恢复96就绪
// //      原因: 泵抽液/排液后状态变100(运动中), 需强停才能恢复96接受下条命令
// //   4. 运动检测: VW4=2→M12.1/M12.2置位(已开始), VW4≠2且已开始→运动完成
// //   5. 运动超时: T102(30秒)防止泵卡在运动态无法退出
// //   6. 全局错误: VW4≥4才报错(VW4=2运动中不算错误)
// // ============================================================
// 
// // 符号说明:
// // VW226 : S3_SubState  S3子状态机
// //          0=进入计算  1=写抽液  2=等抽液运动完成
// //          3=写强停恢复  4=等强停完成+恢复就绪
// //          5=写排液  6=等排液运动完成
// //          7=写强停恢复  8=等强停完成+计算/循环
// //          9=完成转S3.5
// // VD90  : VD_Current_InletVolume 本次进水量(S1差值法结果)
// // VD370 : VD_Vol_Target    目标抽取母液体积(μL)
// // VD372 : VD_Remaining_Vol 本轮剩余待加药量(μL),S3进入时=VD_Vol_Target
// // VD102 : VD_Dose_Steps    本次循环目标步数(REAL)
// // VW204 : MB_Pump_Aspirate 抽液步数缓冲(映射40006)
// // VW206 : MB_Pump_Dispense 排液步数缓冲(映射40007)
// // VD232 : PumpWrite_Addr   FC06写目标Modbus地址
// // VW230 : PumpWrite_Data   FC06写数据
// // M11.6 : PumpWrite_Req    写请求(FC13置位,FC4执行后清零)
// // M11.7 : PumpWrite_Busy   写忙标志(FC4管理)
// // M12.0 : PumpWrite_Done   写完成(FC4置位,FC13清零)
// // M12.1 : Pump_Asp_Started 抽液运动已开始(VW4曾=2)
// // M12.2 : Pump_Disp_Started 排液运动已开始(VW4曾=2)
// // V303.4: M_Alarm_SyringePump 注射泵通讯/动作异常
// // VW4   : 注射泵归一化状态码(0=就绪96,1=空闲64,2=运动中100,≥4=错误)
// // VD346 : 运算中间变量(避免污染HMI设定区)
// // T102  : 运动超时定时器(30秒,子状态2/6复用)
// 
// 
BEGIN
Network 1
//  S3进入/子状态0 - 计算目标加药量,初始化剩余量,启动潜水泵搅拌,清握手位
//  仅在VW226=0时执行一次(FC12进入S3时已清VW226=0)
LD     Always_On:SM0.0
AW=    VW226, 0
LPS
// ? v2.0 浓度参数删除: 目标加药量由用户直接输入VD370(HMI设定),不再通过浓度×水量/母液浓度 公式计算
 // ? v2.0 浓度参数删除: 目标加药量由用户直接输入VD370(HMI设定),不再通过浓度×水量/母液浓度 公式计算
//    原公式: VD346 = VD10(浓度) × VD90(本次进水量) / VD14(母液浓度)
 //    原公式: VD346 = VD10(浓度) × VD90(本次进水量) / VD14(母液浓度)
MOVR   VD370, VD372          // VD_Remaining_Vol = 用户设定的目标加药量
// S3期间保持潜水泵运行(搅拌+加药同时进行)
   // S3期间保持潜水泵运行(搅拌+加药同时进行)
S      CPU_输出0:Q0.0, 1
S      CPU_输出1:Q0.1, 1
// 清写握手位,避免上一周期残留误判
         // 清写握手位,避免上一周期残留误判
R      M12.0, 1
R      M12.1, 1
R      M12.2, 1
R      M11.6, 1
R      M11.7, 1
R      T102, 1
MOVW   1, VW226              // 进入子状态1:计算并写抽液步数
LPP




Network 2
//  S3全局错误检测 - 注射泵通讯/动作异常或状态码报错(≥4)
//  注: VW4=2(运动中)不算错误,不会触发此检测
LD     V303.4                // FC4已置位的通讯/动作故障
LD     Always_On:SM0.0
AW=    VW2, 3
AW>=   VW4, 4                // 状态码≥4(归一化错误码,不含运动中)
OLD
LPS
R      CPU_输出0:Q0.0, 1       // 停潜水泵1
R      CPU_输出1:Q0.1, 1       // 停潜水泵2
S      V303.4, 1             // 确保报警位
MOVW   99, VW2               // 转S_ERROR
MOVW   0, VW226              // 清子状态
R      M12.0, 1
R      M12.1, 1
R      M12.2, 1
R      M11.6, 1
R      M11.7, 1
R      T102, 1
LPP




Network 3
//  子状态1 - 计算本次循环步数并下发抽液指令(16#9C46)
//  条件: 无进行中的写请求/写忙/写完成
LD     Always_On:SM0.0
AW=    VW226, 1
AN     M11.6
AN     M11.7
AN     M12.0
// 计算本次循环步数 = VD_Remaining_Vol / VD_StepResolution
 // 计算本次循环步数 = VD_Remaining_Vol / VD_StepResolution
MOVR   VD372, VD346          // VD346 = VD_Remaining_Vol(μL)
/R     VD350, VD346          // VD346 = steps(REAL)
// 限制最大6000步(25ml注射器容量)
     // 限制最大6000步(25ml注射器容量)
LD     Always_On:SM0.0
AR>=   VD346, 6000.0         // steps >= 6000 ?
JMP    20                    // 是 -> 限制为6000
ROUND  VD346, AC0
MOVR   AC0, VD102            // VD_Dose_Steps < 6000
JMP    21                    // 跳过限制分支
LBL    20
MOVR   6000.0, VD102         // 限制为6000步
LBL    21
// 检查步数有效性(ROUND后剩余量不足一步时直接完成)
 // 检查步数有效性(ROUND后剩余量不足一步时直接完成)
ROUND  VD102, AC0
LD     Always_On:SM0.0
AR<=   AC0, 0.0              // 本次循环步数 <= 0 ?
JMP    22                    // 是 -> 直接转完成
// 同步写入抽/排液步数缓冲(供HMI/调试查看)
  // 同步写入抽/排液步数缓冲(供HMI/调试查看)
MOVW   AC0, VW204
MOVW   AC0, VW206
// 重新建立执行条件后下发抽液指令
          // 重新建立执行条件后下发抽液指令
// ★泵就绪(VW4=0)才允许写, 避免运动中下发导致异常码4
 // ★泵就绪(VW4=0)才允许写, 避免运动中下发导致异常码4
LD     Always_On:SM0.0
AW=    VW226, 1
AN     M11.6
AN     M11.7
AN     M12.0
AW=    VW4, 0
MOVW   AC0, VW230            // 写数据=本次循环步数
MOVD   16#9C46, VD232        // ★十六进制地址(40006=16#9C46)
S      M11.6, 1              // 置写请求
JMP    23
LBL    22
// 剩余量不足一步,无需再加药,直接转完成
      // 剩余量不足一步,无需再加药,直接转完成
MOVW   9, VW226
LBL    23




Network 4
//  子状态1 - 抽液写完成处理
LD     M12.0
AW=    VW226, 1
LPS
A      V303.4                // 写失败(FC4已置报警)
R      CPU_输出0:Q0.0, 1
R      CPU_输出1:Q0.1, 1
MOVW   99, VW2
MOVW   0, VW226
R      M12.0, 1
R      M11.6, 1
R      M11.7, 1
R      T102, 1
LPP
LD     M12.0
AW=    VW226, 1
AN     V303.4                // 写成功
R      M12.0, 1
R      M11.6, 1
MOVW   2, VW226              // →子状态2:等抽液运动完成




Network 5
//  子状态2 - 等待抽液运动完成
//  T102: 30秒超时(防止泵卡在运动态)
//  M12.1: 抽液运动已开始(VW4曾=2)
//  完成: (M12.1=1 AND VW4≠2) OR T102超时 → 子状态3(写强停)
//  T102运行(仅在子状态2时计时)
LD     Always_On:SM0.0
AW=    VW226, 2
TON    T102, 300             // 30秒(300×100ms)


// 检测运动开始: VW4=2 → 置M12.1
   // 检测运动开始: VW4=2 → 置M12.1
LD     Always_On:SM0.0
AW=    VW226, 2
AW=    VW4, 2
S      M12.1, 1


// 运动完成: M12.1=1 AND VW4≠2 → 子状态3(写强停恢复)
 // 运动完成: M12.1=1 AND VW4≠2 → 子状态3(写强停恢复)
LD     M12.1
AW=    VW226, 2
AW<>   VW4, 2
R      T102, 1
R      M12.1, 1
MOVW   3, VW226


// 超时: T102 → 强制子状态3(强停恢复,防止卡死)
 // 超时: T102 → 强制子状态3(强停恢复,防止卡死)
LD     T102
AW=    VW226, 2
R      T102, 1
R      M12.1, 1
MOVW   3, VW226




Network 6
//  子状态3 - 下发强停指令(16#9C42=1)恢复96就绪
//  ★强停无需就绪门控: 用于紧急停止/恢复, 不检查VW4=0
LD     Always_On:SM0.0
AW=    VW226, 3
AN     M11.6
AN     M11.7
AN     M12.0
LPS
MOVW   1, VW230              // 强停数据=1
MOVD   16#9C42, VD232        // ★十六进制地址(40002=16#9C42)
S      M11.6, 1              // 置写请求
LPP




Network 7
//  子状态3 - 强停写完成处理
LD     M12.0
AW=    VW226, 3
LPS
A      V303.4                // 写失败
R      CPU_输出0:Q0.0, 1
R      CPU_输出1:Q0.1, 1
MOVW   99, VW2
MOVW   0, VW226
R      M12.0, 1
R      M11.6, 1
R      M11.7, 1
LPP
LD     M12.0
AW=    VW226, 3
AN     V303.4                // 写成功
R      M12.0, 1
R      M11.6, 1
MOVW   4, VW226              // →子状态4:等恢复就绪




Network 8
//  子状态4 - 等待泵恢复就绪(VW4=0=96就绪态)
//  强停后泵从100→96, 需等待VW4回到0才能接受下一条命令
LD     Always_On:SM0.0
AW=    VW226, 4
AW=    VW4, 0
MOVW   5, VW226              // →子状态5:写排液步数




Network 9
//  子状态5 - 下发排液指令(16#9C47)
//  ★泵就绪(VW4=0)才允许写, 避免运动中下发导致异常码4
LD     Always_On:SM0.0
AW=    VW226, 5
AN     M11.6
AN     M11.7
AN     M12.0
AW=    VW4, 0
LPS
ROUND  VD102, AC0
MOVW   AC0, VW230
MOVW   AC0, VW206
MOVD   16#9C47, VD232        // ★十六进制地址(40007=16#9C47)
S      M11.6, 1
LPP




Network 10
//  子状态5 - 排液写完成处理
LD     M12.0
AW=    VW226, 5
LPS
A      V303.4
R      CPU_输出0:Q0.0, 1
R      CPU_输出1:Q0.1, 1
MOVW   99, VW2
MOVW   0, VW226
R      M12.0, 1
R      M11.6, 1
R      M11.7, 1
R      T102, 1
LPP
LD     M12.0
AW=    VW226, 5
AN     V303.4
R      M12.0, 1
R      M11.6, 1
MOVW   6, VW226              // →子状态6:等排液运动完成




Network 11
//  子状态6 - 等待排液运动完成
//  (逻辑同子状态2, 使用M12.2替代M12.1)
LD     Always_On:SM0.0
AW=    VW226, 6
TON    T102, 300             // 30秒


LD     Always_On:SM0.0
AW=    VW226, 6
AW=    VW4, 2
S      M12.2, 1


// 运动完成: M12.2=1 AND VW4≠2 → 子状态7(写强停恢复)
 // 运动完成: M12.2=1 AND VW4≠2 → 子状态7(写强停恢复)
LD     M12.2
AW=    VW226, 6
AW<>   VW4, 2
R      T102, 1
R      M12.2, 1
MOVW   7, VW226


// 超时: T102 → 强制子状态7
        // 超时: T102 → 强制子状态7
LD     T102
AW=    VW226, 6
R      T102, 1
R      M12.2, 1
MOVW   7, VW226




Network 12
//  子状态7 - 下发强停指令(16#9C42=1)恢复96就绪
//  ★强停无需就绪门控: 用于紧急停止/恢复, 不检查VW4=0
LD     Always_On:SM0.0
AW=    VW226, 7
AN     M11.6
AN     M11.7
AN     M12.0
LPS
MOVW   1, VW230
MOVD   16#9C42, VD232
S      M11.6, 1
LPP




Network 13
//  子状态7 - 强停写完成处理
LD     M12.0
AW=    VW226, 7
LPS
A      V303.4
R      CPU_输出0:Q0.0, 1
R      CPU_输出1:Q0.1, 1
MOVW   99, VW2
MOVW   0, VW226
R      M12.0, 1
R      M11.6, 1
R      M11.7, 1
LPP
LD     M12.0
AW=    VW226, 7
AN     V303.4
R      M12.0, 1
R      M11.6, 1
MOVW   8, VW226              // →子状态8:等恢复就绪+计算/循环




Network 14
//  子状态8 - 等待泵恢复就绪 + 计算本轮体积 + 判断循环/完成
//  等待VW4=0(就绪), 然后计算本轮排出药量, 判断是否完成全部加药量
LD     Always_On:SM0.0
AW=    VW226, 8
AW=    VW4, 0
LPS
// 计算本次循环实际排出药量 = VD_Dose_Steps × VD_StepResolution
 // 计算本次循环实际排出药量 = VD_Dose_Steps × VD_StepResolution
MOVR   VD102, AC0            // AC0 = 本次循环步数(REAL)
*R     VD350, AC0            // AC0 = 本次循环体积(μL)
// 累加本次循环排出药量到累计加药量
         // 累加本次循环排出药量到累计加药量
+R     AC0, VD440            // VD_Dosed_Volume_Total += 本次循环体积
// 扣减剩余待加药量
                 // 扣减剩余待加药量
-R     AC0, VD372            // VD_Remaining_Vol -= 本次循环体积
LPP
// 判断是否完成全部加药量(与恢复就绪条件AND)
  // 判断是否完成全部加药量(与恢复就绪条件AND)
AR>=   VD440, VD370          // 累计加药量 >= 目标量 ?
JMP    30                    // 是 -> 完成
// 未完成: 清本轮握手位,返回子状态1继续下一轮
  // 未完成: 清本轮握手位,返回子状态1继续下一轮
LD     Always_On:SM0.0
AW=    VW226, 8
AW=    VW4, 0
AR<    VD440, VD370          // 确认未完成
R      M12.0, 1
R      M12.1, 1
R      M12.2, 1
R      M11.6, 1
R      M11.7, 1
MOVW   1, VW226              // 返回子状态1:下一轮抽液
JMP    31
LBL    30
// 完成: 转子状态9
                // 完成: 转子状态9
LD     Always_On:SM0.0
AW=    VW226, 8
MOVW   9, VW226
LBL    31




Network 15
//  子状态9 - S3完成,停潜水泵,转S3.5
LD     Always_On:SM0.0
AW=    VW226, 9
LPS
R      CPU_输出0:Q0.0, 1
R      CPU_输出1:Q0.1, 1
R      M12.0, 1
R      M12.1, 1
R      M12.2, 1
R      M11.6, 1
R      M11.7, 1
R      T102, 1
MOVW   0, VW226
MOVW   4, VW2                // VW2=4(S3.5)
LPP




// ============================================================
 // ============================================================
// 文件结束
                     // 文件结束
// 说明:
                      // 说明:
//   1. 采用VW226子状态机(0~9),抽液/排液分两步下发,每步等待FC4写完成(M12.0)
 //   1. 采用VW226子状态机(0~9),抽液/排液分两步下发,每步等待FC4写完成(M12.0)
//   2. 每次抽液/排液运动完成后发强停(40002=1)恢复96就绪态:
 //   2. 每次抽液/排液运动完成后发强停(40002=1)恢复96就绪态:
//      抽液→等运动→强停→等就绪→排液→等运动→强停→等就绪→计算/循环
 //      抽液→等运动→强停→等就绪→排液→等运动→强停→等就绪→计算/循环
//   3. 运动检测: VW4=2(100运动中)→M12.1/M12.2置位,VW4≠2且已运动→运动完成
 //   3. 运动检测: VW4=2(100运动中)→M12.1/M12.2置位,VW4≠2且已运动→运动完成
//   4. 运动超时: T102(30秒)防止泵卡在运动态,T102超时直接发强停恢复
 //   4. 运动超时: T102(30秒)防止泵卡在运动态,T102超时直接发强停恢复
//   5. 支持多次抽液+排液循环:单循环步数限制6000步(25ml注射器容量),
 //   5. 支持多次抽液+排液循环:单循环步数限制6000步(25ml注射器容量),
//      每次排液后强停恢复→累加实际体积到VD378并扣减VD372,直到累计>=目标量
 //      每次排液后强停恢复→累加实际体积到VD378并扣减VD372,直到累计>=目标量
//   6. 全局错误: VW4≥4(不含VW4=2运动中)或V303.4立即转S_ERROR并安全停泵
 //   6. 全局错误: VW4≥4(不含VW4=2运动中)或V303.4立即转S_ERROR并安全停泵
//   7. S3期间Q0.0/Q0.1保持运行,完成/出错时停止
 //   7. S3期间Q0.0/Q0.1保持运行,完成/出错时停止
//   8. 所有Modbus地址使用十六进制格式(16#9C46/16#9C47/16#9C42)
 //   8. 所有Modbus地址使用十六进制格式(16#9C46/16#9C47/16#9C42)
//      避免十进制大数被解析为INT导致MBUS_MSG Error=6
 //      避免十进制大数被解析为INT导致MBUS_MSG Error=6
// ============================================================
 // ============================================================


END_SUBROUTINE_BLOCK

SUBROUTINE_BLOCK State_S35_Rest:SBR9
TITLE=// ============================================================
// // 文件: FC14_State_S35_Rest.stl
// // 功能: S3.5静止等候 (VW2=4)
// // Story: AQEX-6 状态机骨架 + A2修复(计时转换)
// // 说明: 加药后静止沉降，计时到达VD_RestTime_Target转S4
// // ============================================================
// 
// // 符号说明:
// // VW254 : VD_RestTime_Target×10 转换值(100ms时基,供T39用)
// // VD340 : VD124运算中间变量(避免修改VD_RestTime_Target)
// 
BEGIN
Network 1
//  S3.5进入动作 - 启动计时
//  A2修复: 原骨架标注"待Story1.4补充转换",FC40只输出REAL秒到VD124,
//          从未写入VW294导致T39计时失效。现补转换逻辑。
//  VW294 = VD_RestTime_Target(VD124) × 10 (REAL秒→100ms时基)
LD     Always_On:SM0.0
MOVR   VD124, VD340          // 复制到中间变量(避免修改VD_RestTime_Target)
*R     10.0, VD340
ROUND  VD340, AC0
MOVW   AC0, VW294            // VW254 = VD124×10
R      T39, 1
TON    T39, VW294            // PT=VD_RestTime_Target×10(100ms时基)




Network 2
//  静止等候完成转移至S4
LD     T39                   // 计时到达
MOVW   5, VW2                // VW2=5(S4)




// S3.5无输出动作，仅计时
            // S3.5无输出动作，仅计时
// ============================================================
 // ============================================================
// 文件结束
                     // 文件结束
// 说明:
                      // 说明:
//   1. A2修复: VW254由VD124×10转换写入(原骨架遗漏,导致T39计时失效)
 //   1. A2修复: VW254由VD124×10转换写入(原骨架遗漏,导致T39计时失效)
//   2. VD340为运算中间变量,不污染HMI设定参数
 //   2. VD340为运算中间变量,不污染HMI设定参数
// ============================================================
 // ============================================================


END_SUBROUTINE_BLOCK

SUBROUTINE_BLOCK State_S4_Transfer:SBR10
TITLE=// ============================================================
// // 文件: FC15_State_S4_Transfer.stl
// // 功能: S4上→下转移 (VW2=5)
// // Story: AQEX-6 状态机骨架 + AQEX-7 阀门诊断(已集成) + AQEX-8 节奏纠偏(已集成下缸满计时器清零)
// // v1.1: S4入口增加下缸排空互锁(AN V1.7),静默等待 S6 排空后自动开阀
// // v1.2: 新增 S4 等待计时(VD_S4Wait_Time)与超时报警(V303.2),用于补偿 S4 等待对
// //       VD_S5_Elapsed 的影响,确保下缸有效实验时间严格按 VD_CycleSetpoint 跑满
// // 说明: 开阀B转移,调用FC31阀B诊断(四态诊断+开关到位+超时)
// //       诊断结果VW268: 0进行中/1正常完成/2故障
// //       诊断正常完成 → 清零VD_S5_Elapsed+VD_S4Wait_Time+M10.7(供S5纠偏) → 转S5
// // ============================================================
// 
// // 符号说明:
// // v1.2 新增:
// // VD444 : VD_S4Wait_Time    S4 等待时长(秒), S4 入口 V1.7=1 期间每秒 +1, S4 完成时清零
// // VD448 : VD_S4WaitTimeout  S4 等待超时阈值(秒, 默认 1800=30min, HMI 可调)
// // T61   : S4 等待计时器(100ms 时基, PT=VD_S4WaitTimeout×10)
// // VW286 : VD_S4WaitTimeout×10 转换值(供 T61 用)
// // V303.2: M_Alarm_S4TransferWaitTimeout  S4 等待超时报警(一般级, VW6=49, 仅提示不强制 S_ERROR)
// 
// 
BEGIN
Network 1
//  S4转液动作 + 下缸排空互锁(同NETWORK内,符合S7-200 SMART约束)
//  【业务约束】S4开始前必须确认下缸已排空(V1.7=0)
//    上缸S1~S3.5配液与下缸S6排水可并行(S5预规划不阻塞),
//    仅S4入口检查下缸状态:
//      - 下缸已空(V1.7=0)→ 启动S4转液
//      - 下缸仍满(V1.7=1)→ 等待(不报错、不停机),
//                             每周期轮询直至下缸排空完成
//    S5会在换水周期到时自动转S6排水,本FC每周期检测V1.7,
//    一旦V1.7=0,下一扫描周期自动开阀B转液
//  触发条件: 状态=S4 (VW2=5) 且 下缸=空 (V1.7=0)
//  不用 M10.4 EU:避免首周期V1.7=1时错过启动的隐患
LD     Always_On:SM0.0       // 永真,每周期执行
AW=    VW2, 5                // 仅在S4状态(VW2=5)生效
LPS
AN     V1.7                  // 互锁闸门: V1.7=1(下缸满)屏蔽本段
// 开启阀B + 下缸NC球阀(串联主路,需得电导通)
 // 开启阀B + 下缸NC球阀(串联主路,需得电导通)
S      CPU_输出3:Q0.3, 1
S      CPU_输出6:Q0.6, 1
// 启动S4计时器
                  // 启动S4计时器
R      T40, 1
TON    T40, 32767
// 置上缸状态=空
                  // 置上缸状态=空
R      V1.6, 1
// 启动阀B诊断: 置诊断子状态=1
         // 启动阀B诊断: 置诊断子状态=1
MOVB   1, VB262
MOVB   0, VB263
// 清诊断结果
                    // 清诊断结果
MOVB   0, VB268
MOVB   0, VB269
// 计算VD_Timeout_ValveB(VD362)×10转换值
 // 计算VD_Timeout_ValveB(VD362)×10转换值
MOVR   VD362, VD324
*R     10.0, VD324
ROUND  VD324, AC0
MOVW   AC0, VW274
LPP
// 注: 当V1.7=1(下缸未排空)时,AN V1.7条件为假,本段S/R/计时/赋值指令全部不执行,
 // 注: 当V1.7=1(下缸未排空)时,AN V1.7条件为假,本段S/R/计时/赋值指令全部不执行,
//     FC31(阀B诊断)在NETWORK 2 中仍会被CALL,但因Diag_State_B=0(未启动)而空转,
 //     FC31(阀B诊断)在NETWORK 2 中仍会被CALL,但因Diag_State_B=0(未启动)而空转,
//     故不会产生虚假报警。下缸排空后(V1.7=0),下一周期自动开阀B转液。
 //     故不会产生虚假报警。下缸排空后(V1.7=0),下一周期自动开阀B转液。
// 注: 状态转出S4(VW2≠5)后,本段AW=条件不满足,本段所有动作停止。
 // 注: 状态转出S4(VW2≠5)后,本段AW=条件不满足,本段所有动作停止。




// 【v1.2 新增】S4 等待计时 + 超时报警分支(同 NETWORK 1 内,与转液逻辑并列)
 // 【v1.2 新增】S4 等待计时 + 超时报警分支(同 NETWORK 1 内,与转液逻辑并列)
// 触发条件: 状态=S4 且 V1.7=1(下缸未空,正在等待)
 // 触发条件: 状态=S4 且 V1.7=1(下缸未空,正在等待)
//   - 启动 T61 计时器(100ms 时基, PT=VD_S4WaitTimeout×10)
 //   - 启动 T61 计时器(100ms 时基, PT=VD_S4WaitTimeout×10)
//   - 每秒 VD_S4Wait_Time + 1(由 T62 1s 脉冲驱动)
 //   - 每秒 VD_S4Wait_Time + 1(由 T62 1s 脉冲驱动)
//   - 等待时间 >= 阈值 → 置位 V303.2 + VW6=49(仅提示, 不强制 S_ERROR)
 //   - 等待时间 >= 阈值 → 置位 V303.2 + VW6=49(仅提示, 不强制 S_ERROR)
// 等待期间 AN V1.7 失败(转液已开始),T61 在 NETWORK 3 完成后清零
 // 等待期间 AN V1.7 失败(转液已开始),T61 在 NETWORK 3 完成后清零
LD     Always_On:SM0.0
AW=    VW2, 5                // 仅在S4状态
A      V1.7                  // V1.7=1(下缸满)正在等待
LPS
// 首次进入 S4(V1.7=1)时计算 T61 PT(用 VD_S4WaitTimeout×10)
 // 首次进入 S4(V1.7=1)时计算 T61 PT(用 VD_S4WaitTimeout×10)
LD     Always_On:SM0.0
EU                           // 上升沿(仅首次进入时计算一次)
MOVR   VD448, VD324          // ? Bug A 修复: VD452→VD324 (原VD384是HMI参数ManualDose_Target!)
*R     10.0, VD324
ROUND  VD324, AC0
MOVW   AC0, VW286            // VW286 = VD_S4WaitTimeout×10
LPP
// T61 计时(每周期执行, V1.7=1 期间计时)
 // T61 计时(每周期执行, V1.7=1 期间计时)
LD     Always_On:SM0.0
A      V1.7                  // 等待期间持续计时
R      T61, 1
TON    T61, VW286            // PT=VD_S4WaitTimeout×10
// 每秒累加 VD_S4Wait_Time(T62 1s 脉冲)
 // 每秒累加 VD_S4Wait_Time(T62 1s 脉冲)
LD     Always_On:SM0.0
A      V1.7                  // 等待期间
LPS
R      T62, 1
TON    T62, 10               // 1s(10×100ms)
LPP
LD     T62
EU
+R     1.0, VD444            // VD_S4Wait_Time + 1s
R      T62, 1
// 超时报警: T61 到 → 置位 V303.2(报警位), VW6 由 FC3 NETWORK1 统一优先级链计算
 // 超时报警: T61 到 → 置位 V303.2(报警位), VW6 由 FC3 NETWORK1 统一优先级链计算
// ★ 2026-09-11修复: 删除 MOVW 49, VW6(之前因 FC3 错误映射 V303.2→62 而绕过优先级链,
 // ★ 2026-09-11修复: 删除 MOVW 49, VW6(之前因 FC3 错误映射 V303.2→62 而绕过优先级链,
//   现已修正 FC3 为 V303.2→49, 恢复 Story1.6 决策1: 各 FC 只管置位报警位, FC3 统一算 VW6)
 //   现已修正 FC3 为 V303.2→49, 恢复 Story1.6 决策1: 各 FC 只管置位报警位, FC3 统一算 VW6)
LD     T61
S      V303.2, 1             // M_Alarm_S4TransferWaitTimeout
LPP
// 注: 超时报警不强制 S_ERROR, 系统继续等待, 操作员收到 HMI 提示后
 // 注: 超时报警不强制 S_ERROR, 系统继续等待, 操作员收到 HMI 提示后
//     可手动确认/调整 S6 排水, 或修改 VD_S4WaitTimeout
 //     可手动确认/调整 S6 排水, 或修改 VD_S4WaitTimeout
// 注: T61/T62 在 S4 完成时(NETWORK 3)清零; V303.2 在 S4 完成时清零
 // 注: T61/T62 在 S4 完成时(NETWORK 3)清零; V303.2 在 S4 完成时清零


Network 2
//  调用阀B诊断FC31
//  FC31内部处理漫溢保护+四态诊断+开关到位+超时
LD     Always_On:SM0.0
CALL   ValveB_Diag:SBR17




Network 3
//  检查阀B诊断结果
LD     Always_On:SM0.0
LPS
// 诊断正常完成 → 转S5
             // 诊断正常完成 → 转S5
AW=    VW268, 1
R      T40, 1                // 停S4计时
// 记录S4实测时长
                 // 记录S4实测时长
MOVW   T40, VW414            // 暂存定时器值(16位整数)
ITD    VW414, VD444          // 整数→双整数
DTR    VD444, VD74           // 双整数→实数(VD_S4_Actual)
// 置下缸状态=满
                  // 置下缸状态=满
S      V1.7, 1
// 【关键】记录下缸变满时间戳
            // 【关键】记录下缸变满时间戳
LD     Always_On:SM0.0
TODR   VB900
MOVB   VB900, VB10           // DT10 = 当前时间
MOVB   VB901, VB11
MOVB   VB902, VB12
MOVB   VB903, VB13
MOVB   VB904, VB14
MOVB   VB905, VB15
MOVB   VB906, VB16
MOVB   VB908, VB17
// 【Story1.4】下缸变满,清零下缸满计时器+预规划标志(供S5纠偏用)
 // 【Story1.4】下缸变满,清零下缸满计时器+预规划标志(供S5纠偏用)
LD     Always_On:SM0.0
MOVR   0.0, VD178            // VD_S5_Elapsed清零,开始新一轮计时
R      M10.7, 1              // 清预规划触发标志(下轮S5重新触发)
// 【v1.2 新增】S4 等待计时清零(T61/T62/VD_S4Wait_Time/V303.2)
 // 【v1.2 新增】S4 等待计时清零(T61/T62/VD_S4Wait_Time/V303.2)
// 等待时长 VD_S4Wait_Time 已在 NETWORK 1 累加, 此处仅清零, FC16 改用其补偿转 S6 阈值
 // 等待时长 VD_S4Wait_Time 已在 NETWORK 1 累加, 此处仅清零, FC16 改用其补偿转 S6 阈值
LD     Always_On:SM0.0
R      T61, 1                // 停 S4 等待超时计时
R      T62, 1                // 停 S4 等待秒累加计时
MOVR   0.0, VD444            // VD_S4Wait_Time 清零
R      V303.2, 1             // 清 S4 等待超时报警
// 状态转移 S4→S5
               // 状态转移 S4→S5
LD     Always_On:SM0.0
MOVW   6, VW2
LPP




// 注: 漫溢保护、四态诊断、开关到位、超时保护全部由FC31统一处理
 // 注: 漫溢保护、四态诊断、开关到位、超时保护全部由FC31统一处理
// 注: DT时间戳格式需与S7-200 SMART的DT数据类型对齐
 // 注: DT时间戳格式需与S7-200 SMART的DT数据类型对齐
// 注: 断电恢复由FC0统一处理,VW2=5(S4阀B动作中断)时FC0转S_ERROR
 // 注: 断电恢复由FC0统一处理,VW2=5(S4阀B动作中断)时FC0转S_ERROR




// ============================================================
 // ============================================================
// 文件结束
                     // 文件结束
// ============================================================
 // ============================================================
END_SUBROUTINE_BLOCK

SUBROUTINE_BLOCK State_S5_Run:SBR11
TITLE=// ============================================================
// // 文件: FC16_State_S5_Run.stl
// // 功能: S5实验运行中 (VW2=6)
// // Story: AQEX-6 状态机骨架 + AQEX-8 节奏纠偏(已集成)
// // 说明: 下缸满期间累计实验时长,计算Available触发纠偏预规划,
// //       换水周期到转S6排水,实验时长达标转S7结束
// // ============================================================
// 
// // 符号说明:
// // VD150 : VD_Available       剩余可用时间(s) = CycleSetpoint×60 + S6_Rolling - S5_Elapsed
// // VD178 : VD_S5_Elapsed      下缸变满后累计运行秒数(S4完成时清零)
// // VD112 : VD_T_Rolling       滚动实测S1-S3.5总时长(预规划Needed)
// // M10.7 : 预规划已触发标志(本轮只触发一次,转S6/S7时清)
// // VW182 : VW_Corr_Mode       纠偏模式(FC40输入)
// // VW184 : VW_Corr_Result     纠偏结果(FC40输出)
// 
// 
BEGIN
Network 1
//  下缸满计时器 VD_S5_Elapsed 累加
//  每秒VD_S5_Elapsed+1,仅下缸=满期间
LD     Always_On:SM0.0
LPS
A      V1.7                  // 下缸=满才计时
R      T60, 1
TON    T60, 10               // 1秒(10×100ms)
LPP
LD     T60                   // 1秒到
EU
+R     1.0, VD178            // VD_S5_Elapsed + 1
R      T60, 1                // 重置进入下一秒
// 注: 断电恢复时VD_S5_Elapsed由FC0_SysInit用RTC重算(Story 1.7完善)
 // 注: 断电恢复时VD_S5_Elapsed由FC0_SysInit用RTC重算(Story 1.7完善)




Network 2
//  Available计算 + 预规划上升沿触发(转S1上缸配液)
//  VD_Available = VD_CycleSetpoint×60 + VD_S6_Rolling - VD_S5_Elapsed
LD     Always_On:SM0.0
MOVR   VD354, VD150          // VD_CycleSetpoint(min)
*R     60.0, VD150           // →秒
+R     VD116, VD150          // + VD_S6_Rolling
-R     VD178, VD150          // - VD_S5_Elapsed = VD_Available


// 预规划上升沿: Available <= VD_T_Rolling 且 本轮未触发过
 // 预规划上升沿: Available <= VD_T_Rolling 且 本轮未触发过
LD     Always_On:SM0.0
LPS
AR<=   VD150, VD112          // Available <= T_Rolling ?
AN     M10.7                 // 且本轮未触发过
S      M10.7, 1              // 锁存:本轮已触发
// 填入FC40输入: 模式=0(预规划), Needed=VD_T_Rolling
 // 填入FC40输入: 模式=0(预规划), Needed=VD_T_Rolling
MOVW   0, VW182
MOVR   VD112, VD154          // Needed = VD_T_Rolling
CALL   RhythmCorrection:SBR19
// 检查纠偏结果: 非"人工介入(4)"才启动S1
  // 检查纠偏结果: 非"人工介入(4)"才启动S1
LPS
AW<>   VW184, 4
LPS
AN     V1.6                  // 上缸=空(正常)
MOVW   1, VW2                // →S1启动新一轮上缸配液
LPP
LPP
LPP


// 预规划触发后上缸≠空(异常:上一轮S4未排空)
  // 预规划触发后上缸≠空(异常:上一轮S4未排空)
LD     M10.7
A      V1.6                  // 上缸=满(异常)
S      V301.6, 1             // 报警(上缸未排空异常)
MOVW   99, VW2




Network 3
//  实验时长累加(仅下缸=满期间)
//  VD_ExperimentDuration_Accum(VD366)每分钟+1
LD     V1.7                  // 下缸=满
R      T47, 1
TON    T47, 600              // 60秒(600×100ms)
LD     T47                   // 1分钟到
EU
+R     1.0, VD366            // VD_ExperimentDuration_Accum + 1(分钟)




Network 4
//  换水周期到达 - 转S6排水
//  v1.2: VD_S5_Elapsed >= VD_CycleSetpoint×60 - VD_S4Wait_Time
//        即: 实际下缸满的有效时长 >= 用户期望的实验周期
//        (V1.7=1 期间被 S4 等待占用的时间, 在 S4 完成时已清零 VD_S5_Elapsed,
//         但用户期望的下缸满实验时长是 VD_CycleSetpoint, 此处通过阈值补偿保证
//         实际下缸"有效"实验时间严格按 VD_CycleSetpoint 跑满)
LD     Always_On:SM0.0
LPS
MOVR   VD354, AC0            // VD_CycleSetpoint(min)
*R     60.0, AC0             // →秒
-R     VD444, AC0            // v1.2: 减去 S4 等待时长(VD_S4Wait_Time)
AR>=   VD178, AC0            // 已满时长 >= 换水周期(补偿后) ?
R      M10.7, 1              // 清预规划触发标志(下轮重新触发)
R      T60, 1                // 停下缸满计时器
MOVW   7, VW2                // →S6排水(VW2=7)
LPP




Network 5
//  实验时长达标 - 转S7实验结束
//  VD_ExperimentDuration_Accum >= VD_ExperimentTarget → 实验结束
LD     Always_On:SM0.0
LPS
AR>=   VD366, VD24           // 累计时长 >= 目标时长
R      T41, 1                // 停周期计时
R      T60, 1                // 停下缸满计时器
R      M10.7, 1              // 清预规划触发标志
MOVW   8, VW2                // →S7(VW2=8)
LPP




Network 6
//  HMI手动停止命令
LD     V0.2                  // CMD_Stop
EU
R      T41, 1
R      T60, 1
R      M10.7, 1              // 清预规划触发标志
MOVW   8, VW2                // →S7(VW2=8)
S      V1.2, 1               // STA_StopAck握手
R      V0.2, 1               // 清停止命令




// 注: 纠偏预规划由FC40完成,二次校正由FC11(S1完成)调用FC40
 // 注: 纠偏预规划由FC40完成,二次校正由FC11(S1完成)调用FC40
// 注: S5与S1-S3.5并行:预规划触发转S1开始上缸配液,下缸继续实验至换水周期到转S6
 // 注: S5与S1-S3.5并行:预规划触发转S1开始上缸配液,下缸继续实验至换水周期到转S6
// 注: 断电恢复VD_S5_Elapsed重算由FC0_SysInit负责(Story 1.7)
 // 注: 断电恢复VD_S5_Elapsed重算由FC0_SysInit负责(Story 1.7)
// 注: 断电恢复由FC0统一处理,VW2=6(S5无阀门动作)时FC0保持S5并重算VD_S5_Elapsed
 // 注: 断电恢复由FC0统一处理,VW2=6(S5无阀门动作)时FC0保持S5并重算VD_S5_Elapsed
// 注: 上缸配液完成后若下缸仍未到换水周期,状态停留逻辑由FC14(S3.5)细化(后续Story)
 // 注: 上缸配液完成后若下缸仍未到换水周期,状态停留逻辑由FC14(S3.5)细化(后续Story)




// ============================================================
 // ============================================================
// 文件结束
                     // 文件结束
// ============================================================
 // ============================================================
END_SUBROUTINE_BLOCK

SUBROUTINE_BLOCK State_S6_Drain:SBR12
TITLE=// ============================================================
// // 文件: FC17_State_S6_Drain.stl
// // 功能: S6下缸排水 (VW2=7)
// // Story: AQEX-6 状态机骨架 + AQEX-7 阀门诊断(已集成)
// // 说明: 开阀C排水，调用FC32阀C诊断(四态诊断+开关到位+超时)
// //       诊断结果VW270: 0进行中/1正常完成/2故障
// // ============================================================
// 
// // 符号说明:
// // VW264 : Diag_State_C  阀C诊断子状态
// // VW270 : Diag_Result_C 阀C诊断结果
// // VW276 : VD_Timeout_ValveC×10 转换值(供FC32用)
// 
// 
BEGIN
Network 1
//  S6首次进入动作
LD     M10.7                 // S6首次进入脉冲
EU
LPS
// 开启阀C
                     // 开启阀C
S      CPU_输出4:Q0.4, 1
// 启动S6计时器
                  // 启动S6计时器
R      T42, 1
TON    T42, 32767
// 启动阀C诊断: 置诊断子状态=1
         // 启动阀C诊断: 置诊断子状态=1
MOVB   1, VB264
MOVB   0, VB265
// 清诊断结果
                    // 清诊断结果
MOVW   0, VW270
// 计算VD_Timeout_ValveC(VD54)×10转换值
 // 计算VD_Timeout_ValveC(VD54)×10转换值
MOVR   VD54, VD328
*R     10.0, VD328
ROUND  VD328, AC0
MOVW   AC0, VW276
LPP




Network 2
//  调用阀C诊断FC32
//  FC32内部处理四态诊断+开关到位+超时(阀C无漫溢保护)
LD     Always_On:SM0.0
CALL   ValveC_Diag:SBR18




Network 3
//  检查阀C诊断结果
LD     Always_On:SM0.0
LPS
// 诊断正常完成 → 排水完成处理
          // 诊断正常完成 → 排水完成处理
AW=    VW270, 1
R      T42, 1                // 停S6计时
// 记录S6实测时长
                 // 记录S6实测时长
MOVW   T42, VW414            // 暂存定时器值(16位整数)
ITD    VW414, VD444          // 整数→双整数
DTR    VD444, VD78           // 双整数→实数(VD_S6_Actual)
// 更新VD_S6_Rolling(滚动实测)
    // 更新VD_S6_Rolling(滚动实测)
MOVR   VD78, VD116           // VD_S6_Rolling
// 置下缸状态=空
                  // 置下缸状态=空
R      V1.7, 1
LPP




Network 4
//  排水后状态转移
//  若实验未结束(换水周期内) → 返回S5
//  若实验已结束(M10.6标志) → 转S7
LD     Always_On:SM0.0
LPS
AN     M10.6                 // 实验未结束
MOVW   6, VW2                // 返回S5
LPP


LD     M10.6                 // 实验已结束
R      M10.6, 1
MOVW   8, VW2                // 转S7




// 注: 四态诊断、开关到位、超时保护全部由FC32统一处理
 // 注: 四态诊断、开关到位、超时保护全部由FC32统一处理
// 注: VD_S6_Rolling滚动平均算法(非直接覆盖)由Story 1.4细化
 // 注: VD_S6_Rolling滚动平均算法(非直接覆盖)由Story 1.4细化




// 注: 断电恢复由FC0统一处理,VW2=7(S6阀C动作中断)时FC0转S_ERROR
 // 注: 断电恢复由FC0统一处理,VW2=7(S6阀C动作中断)时FC0转S_ERROR
// ============================================================
 // ============================================================
// 文件结束
                     // 文件结束
// ============================================================
 // ============================================================


END_SUBROUTINE_BLOCK

SUBROUTINE_BLOCK State_S7_End:SBR13
TITLE=// ============================================================
// // 文件: FC18_State_S7_End.stl
// // 功能: S7实验结束 (VW2=8)
// // Story: AQEX-6 状态机骨架
// // 说明: 实验完成，状态锁定，提示人工按系统复位后回S0
// // ★ v10重大变更: S7彻底屏蔽V0.0(CMD_Start),只响应I0.3(系统复位按钮)
// //   原实现V0.0↑→回S0,但FC10启动还需再按一次,两次按钮才能启动
// //   且V0.0在S7语义不干净(按钮名叫"启动"实际是"清计数器回S0")
// //   改后:S7唯一出口是物理I0.3系统复位按钮,回S0后V0.0正常工作
// //   同时加V301.7周期提示,HMI滚动条显示"请按系统复位"
// // ============================================================
// 
BEGIN
Network 1
//  S7进入动作 - 安全停机
LD     Always_On:SM0.0
// 复位Q0.0~Q0.6(泵/阀),Q0.7/Q8.0报警声光由FC3统一管理,避免与FC3双写导致闪亮
 // 复位Q0.0~Q0.6(泵/阀),Q0.7/Q8.0报警声光由FC3统一管理,避免与FC3双写导致闪亮
R      CPU_输出0:Q0.0, 7       // 泵停、阀A/B/C关,保留Q0.7
// 停止实验时长累加(VD_ExperimentDuration_Accum锁定最终值)
 // 停止实验时长累加(VD_ExperimentDuration_Accum锁定最终值)
R      T47, 1                // 停1分钟基准计时
// 置实验结束标志(供S6判断是否走最终排水→S7路径)
 // 置实验结束标志(供S6判断是否走最终排水→S7路径)
S      M10.6, 1




Network 2
//  ★ v10新增: 周期置位V301.7实验结束提示
//  S7期间每周期置1,HMI滚动条显示"?? 实验已结束,请按【系统复位】按钮后再启动"
//  纯提示位,不加进VW6优先级链,不锁S_ERROR
//  FC10在启动成功时会R V301.7,1,保证状态干净
LD     Always_On:SM0.0
S      V301.7, 1




Network 3
//  ★ v10重写: S7唯一出口 — 物理系统复位按钮I0.3
//  原实现: V0.0↑→回S0 (已删除,改由I0.3负责)
//  复位条件(全部满足):
//    I1.1=OFF 急停已释放(和FC19/S_ERROR复位保持一致)
//    I0.3上升沿 系统复位按钮按下(就地面板物理按钮,非HMI软命令)
//  为什么S7用I0.3不用V0.0:
//    - V0.0语义是"启动实验",在S7里用它回S0是双重语义,不干净
//    - 改后V0.0只在S0有效,按钮语义单一
//    - 物理复位按钮比HMI软命令更安全(实验结束后强制人工确认)
LDN    CPU_输入9:I1.1          // 急停已释放(常闭触点恢复ON=正常)
A      CPU_输入3:I0.3          // 系统复位按钮按下
EU                           // 上升沿(按下瞬间触发一次)
// 清实验结束标志
                  // 清实验结束标志
R      M10.6, 1
// 清握手位(由S0重新管理)
            // 清握手位(由S0重新管理)
R      V1.0, 1
// ★ 顺手清V301.7提示位(HMI滚动条提示消失)
 // ★ 顺手清V301.7提示位(HMI滚动条提示消失)
R      V301.7, 1
// 清零本次实验累计值,准备新一轮
          // 清零本次实验累计值,准备新一轮
MOVR   0.0, VD364            // 清累计流量
MOVR   0.0, VD440            // 清累计加药量
MOVR   0.0, VD372            // 清S3剩余待加药量
// 状态回S0,后续由FC10接管
          // 状态回S0,后续由FC10接管
MOVW   0, VW2




// ============================================================
 // ============================================================
// 文件结束
                     // 文件结束
// ============================================================
 // ============================================================


END_SUBROUTINE_BLOCK

SUBROUTINE_BLOCK State_Error:SBR14
TITLE=// ============================================================
// // 文件: FC19_State_Error.stl
// // 功能: S_ERROR故障锁定 (VW2=99)
// // Story: AQEX-6 状态机骨架 + AQEX-9 急停双通道+安全继电器反馈(详细实现) + AQEX-10 编址修正(V0.5→V0.7)
// // 说明: 急停或最高级报警触发后的故障锁定,强制输出安全状态
// //       继电器故障(V300.5)禁止复位,必须HMI高权限确认(V0.7)+I1.2正常后清除
// // 急停解除(I1.1=OFF,NO 触点释放)+系统复位按钮(I0.3)→回S0  v1.3 改 NO 接法
// // ============================================================
// 
// // 符号说明:
// // I1.1  : DI_EStop           急停反馈(常开 NO,OFF=正常,ON=急停触发)  v1.3 改为接 NO 触点
// // I1.2  : DI_SafetyRelay_FB  安全继电器辅助反馈(ON=动力回路已断开确认)
// // I0.3  : DI_Btn_SystemReset 系统复位按钮(无源常开点动)
// // V0.7  : CMD_SafetyRelayAck HMI高权限确认继电器故障已检修(需二次确认/高权限)
// // V300.4: M_EStop_Latch      急停触发锁存(漫溢级)
// // V300.5: M_Alarm_SafetyRelay 安全继电器故障(最高级)
// // V1.6  : M_TankA_State      上缸状态(0=空,1=满)
// // V1.7  : M_TankB_State      下缸状态(0=空,1=满)
// // VW2   : 状态机状态(FC19写0回S0)
// // VW6   : 报警码
// 
// 
BEGIN
Network 1
//  故障态输出强制安全(与FC2 NETWORK3双保险)
//  S_ERROR态双保险:即使FC2未执行,QB0也强制安全
LD     Always_On:SM0.0
MOVB   0, QB0                // 潜水泵停/阀关/NC电磁阀失电(关闭=安全)
S      CPU_输出7:Q0.7, 1       // 报警声音(FC3管理消音)
// Q8.0灯光由FC3按报警优先级管理(急停/继电器故障=常亮)
 // Q8.0灯光由FC3按报警优先级管理(急停/继电器故障=常亮)




Network 2
//  继电器故障禁止复位检测
//  9.4: 继电器故障不允许任何自动恢复,必须人工检修
//  V300.5=1时,即使I1.1恢复+I0.3按下,也不允许回S0
LD     V300.5                // 继电器故障=1
JMP    1                     // 跳过系统复位,转NETWORK4检查HMI确认
// V300.5=0(无继电器故障) → 继续NETWORK3系统复位
 // V300.5=0(无继电器故障) → 继续NETWORK3系统复位




Network 3
//  急停解除+系统复位按钮 → 回S0
//  复位条件(全部满足):
//    I1.1=OFF(急停按钮已释放,NO 触点恢复)
//    I0.3上升沿(系统复位按钮按下)
//    V300.5=0(NETWORK2已确认无继电器故障)
LDN    CPU_输入9:I1.1          // 急停已释放(常开 NO 触点恢复 OFF)  v1.3 改 NO 接法
A      CPU_输入3:I0.3          // 系统复位按钮按下
EU                           // 上升沿(按下瞬间)
// 清急停锁存
                    // 清急停锁存
R      V300.4, 1             // M_EStop_Latch=0
// 强制上下缸状态置空(9.3:复位后上下缸状态强制置"空")
 // 强制上下缸状态置空(9.3:复位后上下缸状态强制置"空")
R      V1.6, 1               // 上缸=空
R      V1.7, 1               // 下缸=空
// ★ 2026-09-11 新增: 清阀门诊断子状态和计时器
 // ★ 2026-09-11 新增: 清阀门诊断子状态和计时器
// 与OB1停止命令同根因: FC11/FC15/FC17的AW=VW2xx,0前置条件
 // 与OB1停止命令同根因: FC11/FC15/FC17的AW=VW2xx,0前置条件
FILL   0, VW260, 8           // 清 VB260~VB275 (阀A/B/C 诊断)
R      T50, 6                // 清 T50~T55 (阀A/B 诊断计时器)
// 转S0初始化(9.3:回到S0重新开始,不支持从中断点继续)
 // 转S0初始化(9.3:回到S0重新开始,不支持从中断点继续)
MOVW   0, VW2                // VW2=0(S0)
// 清报警码
                     // 清报警码
MOVW   0, VW6
// 停报警声音(灯光由FC3按确认流程管理)
     // 停报警声音(灯光由FC3按确认流程管理)
R      CPU_输出7:Q0.7, 1
JMP    2                     // 复位完成,结束




Network 4
//  继电器故障HMI高权限确认清除
//  9.4: 继电器故障确认需更高权限/二次确认,通过HMI下发V0.7命令
//  V0.7=1表示HMI高权限确认"继电器已检修,动力回路已验证正常"
//  此时要求I1.2=ON(反馈确实正常)才允许清除V300.5
LBL    1
LD     V0.7                  // HMI高权限确认命令(编址修正:V0.5→V0.7)
EU                           // 上升沿(命令下发瞬间)
A      CPU_输入10:I1.2         // 且安全继电器反馈确实正常(已检修)
R      V300.5, 1             // 清除继电器故障报警
R      V0.7, 1               // 清确认命令
// 注: 清除V300.5后,下一周期NETWORK2不再跳过,NETWORK3允许系统复位按钮回S0
 // 注: 清除V300.5后,下一周期NETWORK2不再跳过,NETWORK3允许系统复位按钮回S0
// 注: 若I1.2仍OFF(检修未完成),V300.5保持,不允许清除
 // 注: 若I1.2仍OFF(检修未完成),V300.5保持,不允许清除




Network 5
//  ★ 自动解锁: S_ERROR锁死但所有报警已被自动恢复清除
//  2026-09-11 修复 AQEX-XX: FC3 NETWORK5自动恢复清一般故障报警位
//    (如V301.4阀A开到位超时→I8.0终于ON→FC3自动R V301.4)，
//    导致 VW2=99(状态机锁S_ERROR) + VW6=0(报警清零) 的状态不一致，
//    OB1 NETWORK12按VW6=0计算VB305=0(良好)，掩盖故障。
//  覆盖场景: V301.4/V301.5/V302.0/V302.1/V303.4 等所有可自恢复的一般故障级
//  解锁条件(全部满足):
//    VW2=99(确实锁在S_ERROR) AND VW6=0(报警系统已清零)
//    AND V300.4=0(非急停锁存) AND V300.5=0(非继电器故障)
//    AND I1.1=OFF(急停按钮已释放,NO触点) AND V303.5=0(非RTC丢失)
LDW=   VW2, 99
AW=    VW6, 0
AN     V300.4                // 不是急停锁存
AN     V300.5                // 不是继电器故障
AN     CPU_输入9:I1.1          // 急停按钮已释放(NO触点OFF)
AN     V303.5                // 不是RTC丢失(RTC不会被自动清,保险检查)
// ★ 2026-09-11 新增: 清阀门诊断子状态和计时器(同OB1停止/系统复位根因)
 // ★ 2026-09-11 新增: 清阀门诊断子状态和计时器(同OB1停止/系统复位根因)
FILL   0, VW260, 8
R      T50, 6
MOVW   0, VW2                // 自动回S0
MOVW   0, VW6                // 清报警码
R      CPU_输出7:Q0.7, 1       // 关报警声音
// 注: 不清V1.6/V1.7(缸状态),让FC0/FC10正常处理
 // 注: 不清V1.6/V1.7(缸状态),让FC0/FC10正常处理
// 注: 不碰V300.4/V300.5,上面AN已确认它们为0
 // 注: 不碰V300.4/V300.5,上面AN已确认它们为0
JMP    2                     // → FC19结束




Network 6
//  FC19结束
LBL    2




// 注: 继电器故障(V300.5)优先级最高,禁止系统复位按钮清除
 // 注: 继电器故障(V300.5)优先级最高,禁止系统复位按钮清除
// 注: 继电器故障清除必须HMI高权限V0.7+I1.2双确认,防止误清除
 // 注: 继电器故障清除必须HMI高权限V0.7+I1.2双确认,防止误清除
// 注: 系统复位后上下缸状态强制置空,从S0重新开始(不支持断点续运行)
 // 注: 系统复位后上下缸状态强制置空,从S0重新开始(不支持断点续运行)
// 注: Q8.0报警灯光由FC3统一管理,本FC不操作
 // 注: Q8.0报警灯光由FC3统一管理,本FC不操作




// ============================================================
 // ============================================================
// 文件结束
                     // 文件结束
// ============================================================
 // ============================================================


END_SUBROUTINE_BLOCK

SUBROUTINE_BLOCK ManualControl:SBR15
TITLE=// ============================================================
// // 文件: FC20_ManualControl.stl
// // 功能: 手动控制FC (由OB1仅在S0态调用)
// // Story: AQEX-60 手动控制页
// // 说明:
// //       由OB1在S0态调用；非S0态不调用，避免覆盖其他状态输出
// //       手动命令为脉冲方式(按1松0),由M位锁存输出状态
// //       手动开阀自动打开串联的NC球阀,关阀自动关闭
// // 修复记录:
// //   P1-改为M位锁存,解决FC10每周期清QB0导致手动输出无法保持的问题
// //   P2-NC球阀串联主路,手动开阀时自动打开对应NC阀
// //   P3-【重大修复2026-09-03】手动命令位从V2.4~V3.7迁移至V306.0~V307.3
// //      原地址V2.4~V3.7与VW2(状态机当前状态)物理地址完全重叠(VB2+VB3),
// //      写入任何手动命令位会直接改写VW2,触发非预期状态切换(如V3.1=1→VW2=2→S2预循环→两台泵同时启动)
// //      新地址V306.0~V307.3落在地址表"预留扩展区",与VW2/VW6/VW8等状态/报警字无冲突
// //   P4-【2026-09-03 调试模式】新增V303.5调试模式开关,=1时跳过阀B/阀C的液位联锁(V1.6/V1.7)
// //      联机调试时上下缸无水,V1.6/V1.7=0,导致阀B/阀C手动永远卡死
// //      调试期间V303.5置1可绕过联锁直接开阀;生产前必须V303.5=0(默认)
// // ============================================================
// 
// // 符号表:
// // V306.0 : CMD_Manual_ValveA_Open  手动开阀A   (旧地址V2.4,2026-09-03迁移避开VW2重叠)
// // V306.1 : CMD_Manual_ValveA_Close 手动关阀A   (旧地址V2.5)
// // V306.2 : CMD_Manual_ValveB_Open  手动开阀B   (旧地址V2.6)
// // V306.3 : CMD_Manual_ValveB_Close 手动关阀B   (旧地址V2.7)
// // V306.4 : CMD_Manual_ValveC_Open  手动开阀C   (旧地址V3.0)
// // V306.5 : CMD_Manual_ValveC_Close 手动关阀C   (旧地址V3.1)
// // V306.6 : CMD_Manual_Pump1_On     手动启泵1   (旧地址V3.2)
// // V306.7 : CMD_Manual_Pump1_Off    手动停泵1   (旧地址V3.3)
// // V307.0 : CMD_Manual_Pump2_On     手动启泵2   (旧地址V3.4)
// // V307.1 : CMD_Manual_Pump2_Off    手动停泵2   (旧地址V3.5)
// // V309.0 : M_DebugMode_BypassInterlock 调试模式-跳过液位联锁(0=生产/1=调试,默认0,调试结束后必须清0)
// // V1.6   : STA_TankA_State         上缸液位状态(自动流程FC12置1/FC15清0)
// // V1.7   : STA_TankB_State         下缸液位状态(自动流程FC15/FC16维护)
// // Q0.2   : DO_ValveA 阀A输出
// // Q0.3   : DO_ValveB 阀B输出
// // Q0.4   : DO_ValveC 阀C输出
// // Q0.5   : DO_NCValve_Top NC球阀-上缸(常闭型,得电打开)
// // Q0.6   : DO_NCValve_Bottom NC球阀-下缸(常闭型,得电打开)
// // M13.0  : 阀A手动锁存(=1开阀A,=0关阀A)
// // M13.1  : 阀B手动锁存
// // M13.2  : 阀C手动锁存
// // M13.3  : 泵1手动锁存
// // M13.4  : 泵2手动锁存
// // ============================================================
BEGIN
Network 1
//  手动阀A控制(开/关)
LD     Always_On:SM0.0
A      V306.0
EU
S      M13.0, 1
R      V306.0, 1
LD     Always_On:SM0.0
A      V306.1
EU
R      M13.0, 1
R      V306.1, 1
Network 2
//  手动阀B控制(开/关)
//  联锁条件: 上缸满(V1.6) AND 下缸空(V1.7=0) [生产]
//  调试模式: V309.0=1 跳过联锁(空缸调试用,生产前必须V309.0=0)
LD     Always_On:SM0.0
A      V306.2
EU
LD     V1.6
AN     V1.7
O      V309.0
ALD
S      M13.1, 1
R      V306.2, 1
LD     Always_On:SM0.0
A      V306.3
EU
R      M13.1, 1
R      V306.3, 1
Network 3
//  手动阀C控制(开/关)
//  联锁条件: 下缸满(V1.7) [生产]
//  调试模式: V309.0=1 跳过联锁(空缸调试用,生产前必须V309.0=0)
LD     Always_On:SM0.0
A      V306.4
EU
LD     V1.7
O      V309.0
ALD
S      M13.2, 1
R      V306.4, 1
LD     Always_On:SM0.0
A      V306.5
EU
R      M13.2, 1
R      V306.5, 1
Network 4
//  手动泵1控制(启/停)
LD     Always_On:SM0.0
A      V306.6
EU
S      M13.3, 1
R      V306.6, 1
LD     Always_On:SM0.0
A      V306.7
EU
R      M13.3, 1
R      V306.7, 1
Network 5
//  手动泵2控制(启/停)
LD     Always_On:SM0.0
A      V307.0
EU
S      M13.4, 1
R      V307.0, 1
LD     Always_On:SM0.0
A      V307.1
EU
R      M13.4, 1
R      V307.1, 1
Network 6
//  手动输出映射到Q点
//  在S0态用=线圈覆盖FC10_State_S0_Init中的QB0清零
LD     M13.0
=      CPU_输出2:Q0.2
LD     M13.1
=      CPU_输出3:Q0.3
LD     M13.2
=      CPU_输出4:Q0.4
LD     M13.3
=      CPU_输出0:Q0.0
LD     M13.4
=      CPU_输出1:Q0.1
Network 7
//  NC球阀自动跟随(串联主路,保证手动开阀有水流通)
//  上缸NC阀跟随阀A;下缸NC阀跟随阀B
LD     CPU_输出2:Q0.2
=      CPU_输出5:Q0.5
LD     CPU_输出3:Q0.3
=      CPU_输出6:Q0.6
END_SUBROUTINE_BLOCK

